ARiZoneSkipArea[FormulaFL] := ARiZoneSkipArea[FormulaFL -1] + ARiZoneAreaInt[FormulaFL -1] + ARiAddArmTime[FormulaFL -1];

END_FOR

IF FormulaFL > iRecipeBlockQty THEN
Step:= 2;
ZoneFL := 1;
GroupFL := 1;
END_IF


2:


FOR ZoneFL:= 1 TO iRecipeBlockQty DO

	FOR GroupFL:= 1 TO 10000 DO

		IF GroupFL > ARiZoneSkipArea[ZoneFL] AND GroupFL <= ARiZoneSkipArea[ZoneFL] + ARiZoneAreaInt[ZoneFL] + ARiAddArmTime[ZoneFL]THEN
		Ar10000_iRecipeTimeBlock [GroupFL] := ARiZoneAddress[ZoneFL];
		END_IF

	END_FOR

END_FOR

IF ZoneFL > iRecipeBlockQty AND GroupFL > 10000 THEN
Step:= 3;
END_IF

3:;


END_CASE
*)
CASE Step2 OF

0:;

1:
iSortMFL:=1;

	IF iSortMFL >0 AND iSortMFL <=iRecipeBlockQty THEN
		FOR iSortMFL := 1 TO iRecipeBlockQty DO

			IF iSortMFL = 1 THEN
			AR2SiRecipeTimeBlock[iSortMFL,1] := 1;
			AR2SiRecipeTimeBlock[iSortMFL,2] := ARiZoneAreaInt[iSortMFL] + ARiAddArmTime[iSortMFL];
			AR2SiRecipeTimeBlock[iSortMFL,3] := ARiZoneAddress[iSortMFL];
			END_IF

			IF iSortMFL > 1 THEN
			AR2SiRecipeTimeBlock[iSortMFL,1] := AR2SiRecipeTimeBlock[iSortMFL-1,2]+1;
			AR2SiRecipeTimeBlock[iSortMFL,2] := ARiZoneAreaInt[iSortMFL] + ARiAddArmTime[iSortMFL] +AR2SiRecipeTimeBlock[iSortMFL-1,2] ;
			AR2SiRecipeTimeBlock[iSortMFL,3] := ARiZoneAddress[iSortMFL];
			END_IF

		END_FOR

	END_IF

IF iSortMFL > iRecipeBlockQty THEN
	Step2:=2;
END_IF


2:
iShiftMFL := 1;
iShiftSFL := 1;

	IF iShiftSFL >0 AND iShiftSFL <=iRecipeBlockQty THEN
		FOR iShiftSFL := 1 TO iRecipeBlockQty DO

			IF AR2SiRecipeTimeBlock[iShiftSFL,2] > AR2SiRecipeTimeBlock[iShiftSFL,1]  THEN
			AR2SiRecipeTimeBlock[iShiftMFL,1] := AR2SiRecipeTimeBlock[iShiftSFL,1];
			AR2SiRecipeTimeBlock[iShiftMFL,2] := AR2SiRecipeTimeBlock[iShiftSFL,2];
			AR2SiRecipeTimeBlock[iShiftMFL,3] := AR2SiRecipeTimeBlock[iShiftSFL,3];

							IF iShiftMFL <> iShiftSFL THEN
							AR2SiRecipeTimeBlock[iShiftSFL,1] := 0;
							AR2SiRecipeTimeBlock[iShiftSFL,2] := 0;
							AR2SiRecipeTimeBlock[iShiftSFL,3] := 0;
							END_IF



			iShiftMFL := iShiftMFL + 1;
			END_IF



		END_FOR

	END_IF


IF iShiftSFL > iRecipeBlockQty THEN
	Step2:=3;
END_IF

3:
iClearRemainFL :=1;

	IF iClearRemainFL >0 AND iClearRemainFL <=iRecipeBlockQty THEN
		FOR iClearRemainFL := 1 TO iRecipeBlockQty DO

			IF AR2SiRecipeTimeBlock[iClearRemainFL,2] <= AR2SiRecipeTimeBlock[iClearRemainFL,1]  THEN
			AR2SiRecipeTimeBlock[iClearRemainFL,1] := 0;
			AR2SiRecipeTimeBlock[iClearRemainFL,2] := 0;
			AR2SiRecipeTimeBlock[iClearRemainFL,3] := 0;
			iShiftMFL := iShiftMFL + 1;
			END_IF

		END_FOR


	END_IF

IF iClearRemainFL > iRecipeBlockQty THEN
Step2:=4;
(*Step2:=5;
bCompleted:=TRUE;
*)
END_IF



4:

iAddMFL:=1;

	IF iAddMFL >0 AND iAddMFL <=iRecipeBlockQty THEN
		FOR iAddMFL := 1 TO iRecipeBlockQty DO
(*
		IF AR2SiRecipeTimeBlock[iAddMFL,3] > iStnQty THEN

			IF iAddMFL = 1 THEN
			AR2SiRecipeTimeBlock[iAddMFL,1] := 1;
			AR2SiRecipeTimeBlock[iAddMFL,2] := ARiZoneAreaInt[iAddMFL] + ARiAddArmTime[iAddMFL];
			AR2SiRecipeTimeBlock[iAddMFL,3] := ARiZoneAddress[iAddMFL];
			END_IF

			IF iAddMFL > 1 THEN
			AR2SiRecipeTimeBlock[iAddMFL,1] := AR2SiRecipeTimeBlock[iAddMFL-1,2]+1;
			AR2SiRecipeTimeBlock[iAddMFL,2] := ARiZoneAreaInt[iAddMFL] + ARiAddArmTime[iAddMFL] +AR2SiRecipeTimeBlock[iAddMFL-1,2] ;
			AR2SiRecipeTimeBlock[iAddMFL,3] := ARiZoneAddress[iAddMFL];
			END_IF

		END_IF
*)
		IF AR2SiRecipeTimeBlock[iAddMFL,3] > 0 AND AR2SiRecipeTimeBlock[iAddMFL,3] <= iStnQty THEN

			IF iAddMFL = 1 THEN
			AR2SiRecipeTimeBlock[iAddMFL,1] := 1;
			AR2SiRecipeTimeBlock[iAddMFL,2] := AR2SiRecipeTimeBlock[iAddMFL+1,2];(*ARiZoneAreaInt[iAddMFL] + ARiAddArmTime[iAddMFL] + ARiZoneAreaInt[iAddMFL+1] ;*)
			AR2SiRecipeTimeBlock[iAddMFL,3] := AR2SiRecipeTimeBlock[iAddMFL,3];
			END_IF

			IF iAddMFL > 1 THEN
			AR2SiRecipeTimeBlock[iAddMFL,1] := AR2SiRecipeTimeBlock[iAddMFL-1,1];
			AR2SiRecipeTimeBlock[iAddMFL,2] := AR2SiRecipeTimeBlock[iAddMFL+1,2];(*ARiZoneAreaInt[iAddMFL] + ARiAddArmTime[iAddMFL] +AR2SiRecipeTimeBlock[iAddMFL-1,2] ;*)
			AR2SiRecipeTimeBlock[iAddMFL,3] := AR2SiRecipeTimeBlock[iAddMFL,3];
			END_IF

		END_IF

		END_FOR

	END_IF

IF iAddMFL > iRecipeBlockQty THEN
	Step2:=5;
bCompleted:=TRUE;
END_IF

5:


;
END_CASE

END_FUNCTION_BLOCK

// ---- FBs/B_JKS_NewFB/FBP-StationRelated/fbMainStationProcess.TcPOU
FUNCTION_BLOCK fbMainStationProcess

VAR_INPUT
	(*fbStnSeqProcess*)
	bSavePB_Uni 									: BOOL; 														(*Universal*) (* Input - HMI - Save Push Button on Touchscreen*)
	bLoadPB_Uni 								: BOOL;														(*Universal*) (* Input - HMI - Load Push Button on Touchscreen*)
	bTrackerEn									: BOOL;														(*During Tracker, it will only call arm when process completed*)
	bTrackerBasedOnPreviousTime			: BOOL;

	(*fbGnrStationMasterController*)
	iCurrentStationAddress_Fix 					: INT;															(*Individual*) (* Input - Define current station no so that this fb know which array number to used*)
	iPreCallArmTime_Uni						: INT;															(*Universal*) (* Input - Pre-Call Arm Time, Program will call arm if the Total process timeEV Equal or Lesser than this value*)
	ARbAlternateStnEn : ARRAY [1..iAlternateSetQty] OF BOOL;
	AR2siAlternateStn : ARRAY [1..iAlternateSetQty, 1..iAlternateStnQty] OF INT;


END_VAR

VAR_IN_OUT PERSISTENT

	(*fbStnSeqProcess*)
(*	DsStnSeqProInput_Ind 						: DS_StnSeqProInput;											(*Individual*) (* Input - PV of Instrument (Temperature, pressure, vacuum and etc), Signal of Sensor to allowed program under the current station status.*)
*)	DSStnSeqProcessCtrl_Ind			 		: DS_fbStnSeqProcessCtrl;									(*Individual*) (* InOut - Link with fbStnSeqProcess, so that this fb know the full status of fbStnSeqProcess and determine which action to take*)

	DsStnSeqRepStore_Ind 						: DS_fbStationSequenceRecipeStore; 						(*Individual*) (* InOut - HMI - The full set of DataStructure-StationSequenceRecipe should selectively display on HMI so that user can customise the recipe by choosing/configure the parameters.*)
	DsStnSubRepStore_Ind 						: DS_fbStationSubRecipeStore; 								(*Individual*) (* InOut - HMI - The full set of DataStructure-StationSubRecipe should selectively display on HMI so that user can customise the recipe by choosing/configure the parameters.*)
	DsStnSeqRepCall_Ind 						: DS_fbStationSequenceRecipeCall;							(*Individual*) (* InOut - Used to call StationSequenceRecipe Detail from fbStationSequenceRecipe*)
	DsStnSubRepCall_Ind 						: DS_fbStationSubRecipeCall;								(*Individual*) (* InOut - Used to call StationSubRecipe Detail from fbStationSubRecipe*)

	(*fbGnrStationMasterController*)
	ARbProductRecipeCallEn_Uni 				: ARRAY [0..iStnQty] OF BOOL;					(*Universal*) (* Output - Link with fbGnrProductRecipeMemory, Array based on Current Station No, the fbGnrProductRecipeMemory will start Read info from Memory when this bool turn on*)
	ARiProductRecipeNoCall_Uni 				: ARRAY [0..iStnQty] OF INT;						(*Universal*) (* Output - Link with fbGnrProductRecipeMemory, Array based on Current Station No, the read out from fbGnrProductRecipeMemory is based on this Product Recipe No*)
	ARiProductRecipeStepCall_Uni 				: ARRAY [0..iStnQty] OF INT;						(*Universal*) (* Output - Link with fbGnrProductRecipeMemory, Array based on Current Station No, the read out from fbGnrProductRecipeMemory is based on this Product Recipe Step No*)

	DSfbGnrProductRecipeMemoryOut_Uni 		: DS_fbGnrProductRecipeMemoryOut;						(*Universal*) (* Input - Link with fbGnrProductRecipeMemory, all the read out info from fbGnrProductRecipeMemory will store in this DataStucture*)

	ARbArmReady_Uni							: ARRAY [1..iArmQty] OF BOOL;								(* Universal*) (* Input  - From ArmPnpFB, This signal is used to confirm if the arm is ready and idling*)

	ARiStnNoToCalledArm_Uni					: ARRAY [0..iArmQty] OF INT; 									(*Universal*) (* Output - Link with fbArmPnP, Array based on Arm No, The Int will store which Station that calling the Arm*)
	ARDSGnrFeedArmPnpParameter_Uni		: ARRAY [0..iArmQty] OF DSGnr_CalledArmPnpParameter; 	(*Universal*) (* Output - Link with fbArmPnP, Array based on Current Station No, Arm should move based on this DataStructure Info*)

	DSLdBasketInfo_Uni		 				: DS_BasketInfo;											(*Input - Loading CONFIRM Basket Info*)
	DSUldBasketInfo_Uni		 				: DS_BasketInfo;											(*Input - Uloading CONFIRM Basket Info*)
	ARDsStnBasketInfo_Uni					: ARRAY [1..iStnQty] OF DS_BasketInfo;						(*Input - Station Basket Info*)



END_VAR

VAR_OUTPUT PERSISTENT
	bSaveInd_Uni 								: BOOL; 														(*Universal*) (* Output - HMI - Save Indicator on Touchscreen*)
	bLoadInd_Uni 								: BOOL; 														(*Universal*) (* Output - HMI - Load Indicator on Touchscreen*)
(*	DSStnSeqProOutput_Ind 						:DS_StnSeqProOutput;										(*Individual*) (* Output - To Control Output - When process running, instrument should control by the output in this Data structure*)
*)
END_VAR



VAR PERSISTENT
	(*fbStnSeqProcess*)
	StnSeqProcessfb: fbStnSeqProcess;
	bStnSeqProcessStartInterlock			: BOOL;															(*Individual*) (* Input - Interlocking to Enable the StnSeqProcess Start Signal, It might used on those station with Sliding door for close confirmation before process start*)

	(*fbGnrStationMasterController*)
	GnrStationMasterControllerfb				: fbGnrStationMasterController;
	bStnSeqProcessSt						: BOOL;															(* Output - Link with fbStnSeqProcess, After Read out from fbGnrProductRecipeMemory, this fb will trigger this Bool to start the StnSeqProcess*)
	DSGnrBufferCalledArmPnpParameter 	: DSGnr_CalledArmPnpParameter;								(* Internal used, Buffer Data Structure read out from fbGnrProductRecipeMemory*)
	DSGnrBuffersPnpSequenceDescription	: STRING (99);														(* Internal used, Buffer Description read out from fbGnrProductRecipeMemory*)
	ARiPreviousStnSeqTotalProcessTime 	: ARRAY [0..iProductRecipeArrayQty] OF INT;					(* Internal used, Previous Total Process Time will save into this Array, Array based on StationSequenceNo*)
	iCallStep									: INT;																(* Internal used, to monitor the current Step so that you can indentify the error of this function block if stucked*)
	DSBasketInfo_Ind 							: DS_BasketInfo;												(*Individual*) (* InOut - Basket Information that comes into current station*)

END_VAR
VAR
	bLdStnConfirm: BOOL;
	bUldStnConfirm: BOOL;
	bStn1Confirm: BOOL;
	bGreaterStn1Confirm: BOOL;
	bLesserStnQtyConfirm: BOOL;
	bEqualStnQtyConfirm: BOOL;
	iTotalProcessTimeSV: INT;
END_VAR
VAR // added by the converter: edge detectors and wires of the graphical bodies
    _w1, _w2, _w3 : DS_BasketInfo;
END_VAR

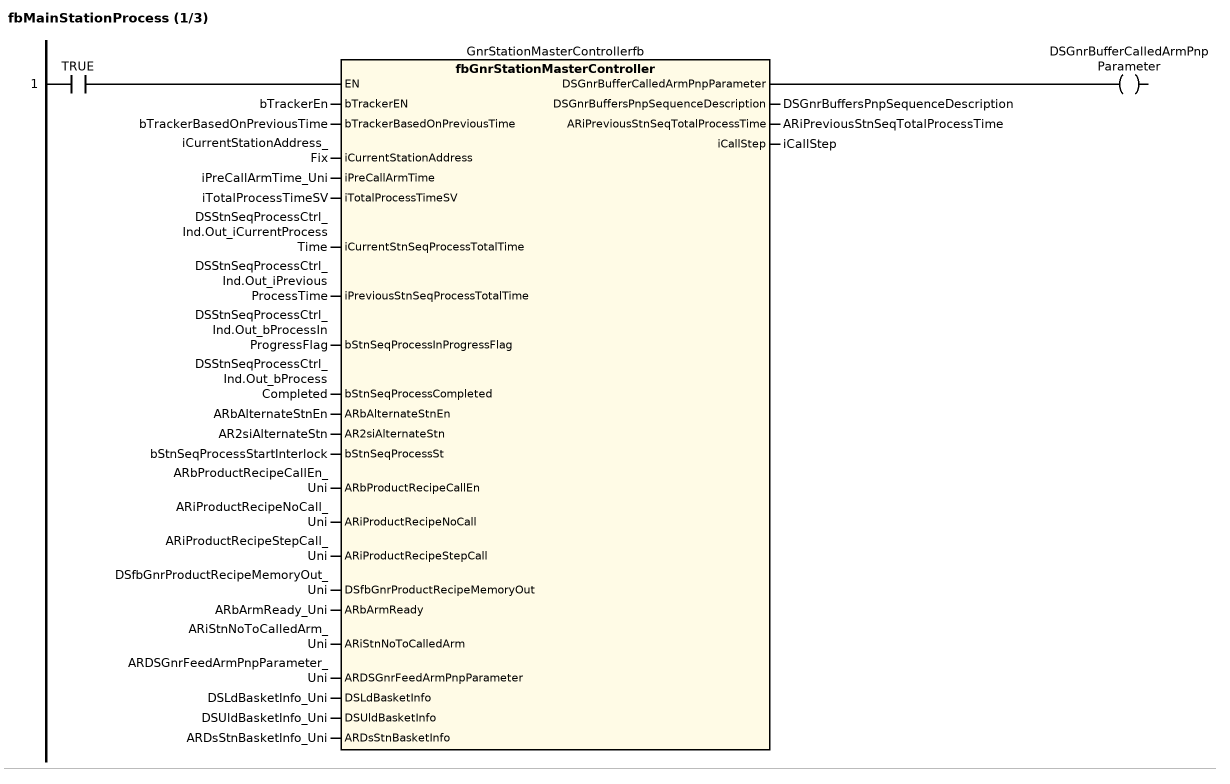
// NETWORK 1
GnrStationMasterControllerfb(
    bTrackerEN := bTrackerEn,
    bTrackerBasedOnPreviousTime := bTrackerBasedOnPreviousTime,
    iCurrentStationAddress := iCurrentStationAddress_Fix,
    iPreCallArmTime := iPreCallArmTime_Uni,
    iTotalProcessTimeSV := iTotalProcessTimeSV,
    iCurrentStnSeqProcessTotalTime := DSStnSeqProcessCtrl_Ind.Out_iCurrentProcessTime,
    iPreviousStnSeqProcessTotalTime := DSStnSeqProcessCtrl_Ind.Out_iPreviousProcessTime,
    bStnSeqProcessInProgressFlag := DSStnSeqProcessCtrl_Ind.Out_bProcessInProgressFlag,
    bStnSeqProcessCompleted := DSStnSeqProcessCtrl_Ind.Out_bProcessCompleted,
    ARbAlternateStnEn := ARbAlternateStnEn,
    AR2siAlternateStn := AR2siAlternateStn,
    bStnSeqProcessSt := bStnSeqProcessStartInterlock,
    ARbProductRecipeCallEn := ARbProductRecipeCallEn_Uni,
    ARiProductRecipeNoCall := ARiProductRecipeNoCall_Uni,
    ARiProductRecipeStepCall := ARiProductRecipeStepCall_Uni,
    DSfbGnrProductRecipeMemoryOut := DSfbGnrProductRecipeMemoryOut_Uni,
    ARbArmReady := ARbArmReady_Uni,
    ARiStnNoToCalledArm := ARiStnNoToCalledArm_Uni,
    ARDSGnrFeedArmPnpParameter := ARDSGnrFeedArmPnpParameter_Uni,
    DSLdBasketInfo := DSLdBasketInfo_Uni,
    DSUldBasketInfo := DSUldBasketInfo_Uni,
    ARDsStnBasketInfo := ARDsStnBasketInfo_Uni,
    DSGnrBuffersPnpSequenceDescription => DSGnrBuffersPnpSequenceDescription,
    ARiPreviousStnSeqTotalProcessTime => ARiPreviousStnSeqTotalProcessTime,
    iCallStep => iCallStep); // fbGnrStationMasterController
DSGnrBufferCalledArmPnpParameter := GnrStationMasterControllerfb.DSGnrBufferCalledArmPnpParameter;

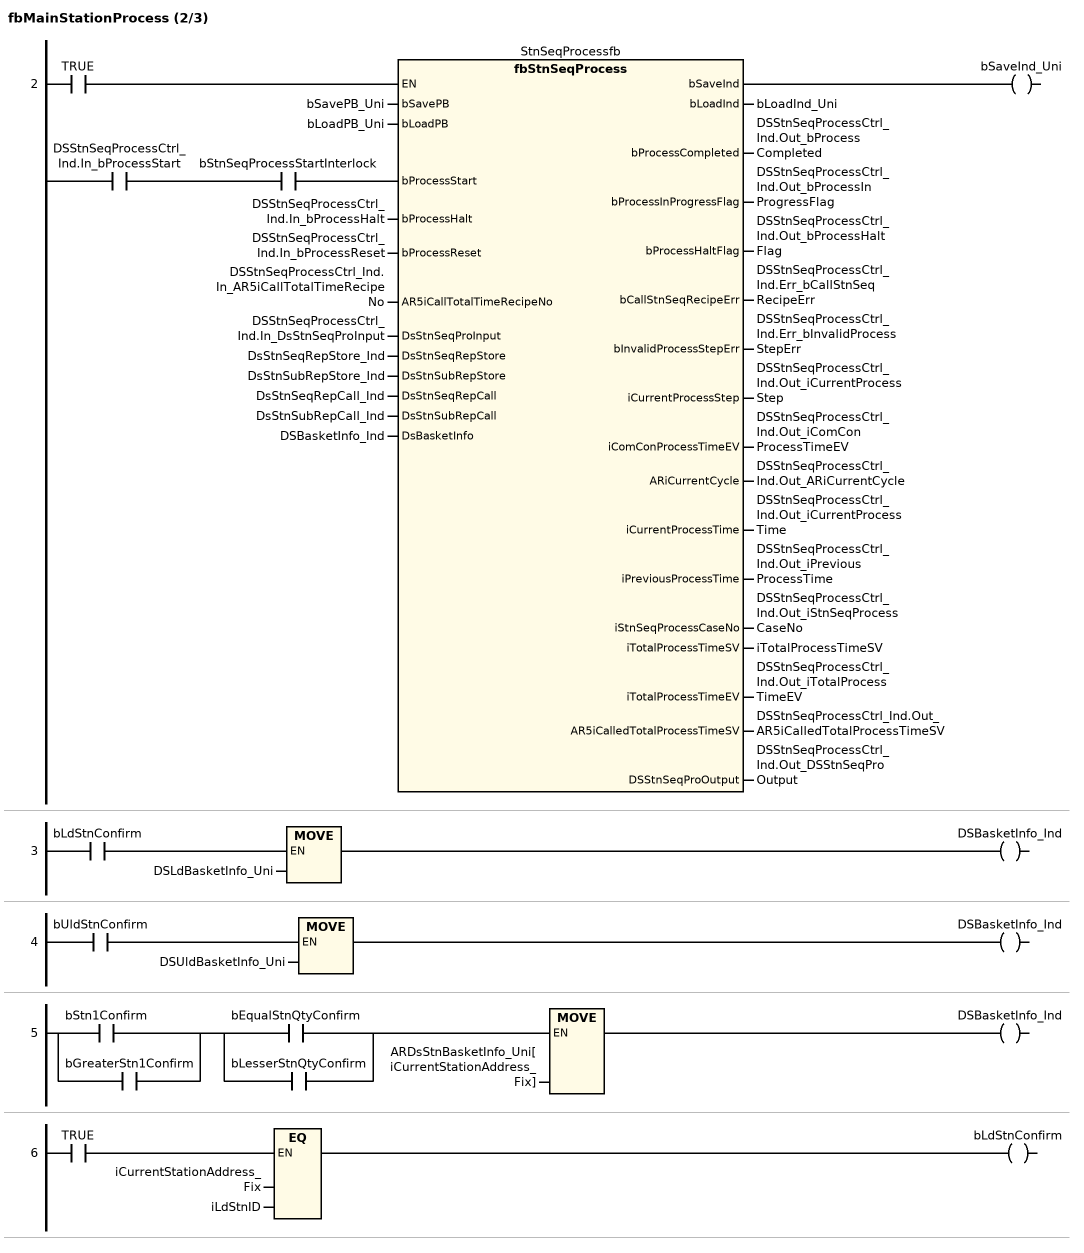
// NETWORK 2
StnSeqProcessfb(
    bSavePB := bSavePB_Uni,
    bLoadPB := bLoadPB_Uni,
    bProcessStart := DSStnSeqProcessCtrl_Ind.In_bProcessStart AND bStnSeqProcessStartInterlock,
    bProcessHalt := DSStnSeqProcessCtrl_Ind.In_bProcessHalt,
    bProcessReset := DSStnSeqProcessCtrl_Ind.In_bProcessReset,
    AR5iCallTotalTimeRecipeNo := DSStnSeqProcessCtrl_Ind.In_AR5iCallTotalTimeRecipeNo,
    DsStnSeqProInput := DSStnSeqProcessCtrl_Ind.In_DsStnSeqProInput,
    DsStnSeqRepStore := DsStnSeqRepStore_Ind,
    DsStnSubRepStore := DsStnSubRepStore_Ind,
    DsStnSeqRepCall := DsStnSeqRepCall_Ind,
    DsStnSubRepCall := DsStnSubRepCall_Ind,
    DsBasketInfo := DSBasketInfo_Ind,
    bLoadInd => bLoadInd_Uni,
    bProcessCompleted => DSStnSeqProcessCtrl_Ind.Out_bProcessCompleted,
    bProcessInProgressFlag => DSStnSeqProcessCtrl_Ind.Out_bProcessInProgressFlag,
    bProcessHaltFlag => DSStnSeqProcessCtrl_Ind.Out_bProcessHaltFlag,
    bCallStnSeqRecipeErr => DSStnSeqProcessCtrl_Ind.Err_bCallStnSeqRecipeErr,
    bInvalidProcessStepErr => DSStnSeqProcessCtrl_Ind.Err_bInvalidProcessStepErr,
    iCurrentProcessStep => DSStnSeqProcessCtrl_Ind.Out_iCurrentProcessStep,
    iComConProcessTimeEV => DSStnSeqProcessCtrl_Ind.Out_iComConProcessTimeEV,
    ARiCurrentCycle => DSStnSeqProcessCtrl_Ind.Out_ARiCurrentCycle,
    iCurrentProcessTime => DSStnSeqProcessCtrl_Ind.Out_iCurrentProcessTime,
    iPreviousProcessTime => DSStnSeqProcessCtrl_Ind.Out_iPreviousProcessTime,
    iStnSeqProcessCaseNo => DSStnSeqProcessCtrl_Ind.Out_iStnSeqProcessCaseNo,
    iTotalProcessTimeSV => iTotalProcessTimeSV,
    iTotalProcessTimeEV => DSStnSeqProcessCtrl_Ind.Out_iTotalProcessTimeEV,
    AR5iCalledTotalProcessTimeSV => DSStnSeqProcessCtrl_Ind.Out_AR5iCalledTotalProcessTimeSV,
    DSStnSeqProOutput => DSStnSeqProcessCtrl_Ind.Out_DSStnSeqProOutput); // fbStnSeqProcess
bSaveInd_Uni := StnSeqProcessfb.bSaveInd;

// NETWORK 3
IF bLdStnConfirm THEN _w1 := DSLdBasketInfo_Uni; END_IF
DSBasketInfo_Ind := _w1;

// NETWORK 4
IF bUldStnConfirm THEN _w2 := DSUldBasketInfo_Uni; END_IF
DSBasketInfo_Ind := _w2;

// NETWORK 5
IF (bStn1Confirm OR bGreaterStn1Confirm) AND (bEqualStnQtyConfirm OR bLesserStnQtyConfirm) THEN
    _w3 := ARDsStnBasketInfo_Uni[iCurrentStationAddress_Fix];
END_IF
DSBasketInfo_Ind := _w3;

// NETWORK 6
bLdStnConfirm := iCurrentStationAddress_Fix = iLdStnID;

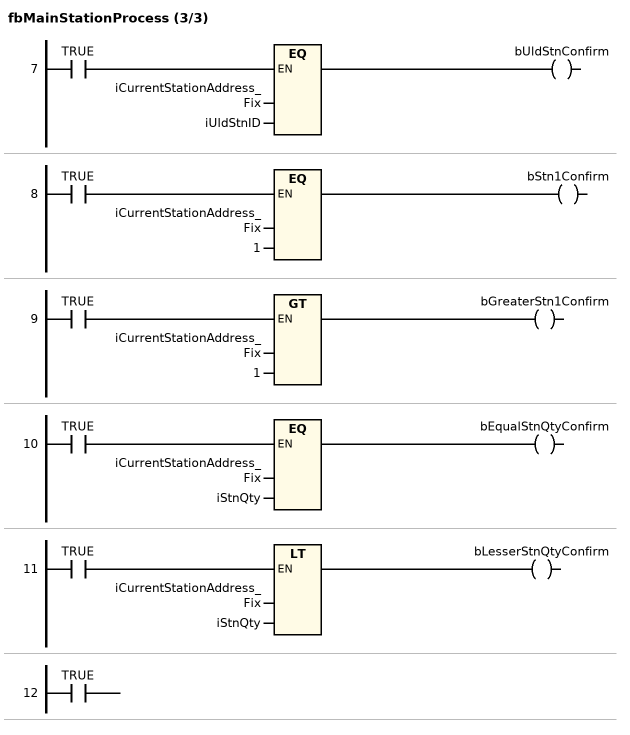
// NETWORK 7
bUldStnConfirm := iCurrentStationAddress_Fix = iUldStnID;

// NETWORK 8
bStn1Confirm := iCurrentStationAddress_Fix = 1;

// NETWORK 9
bGreaterStn1Confirm := iCurrentStationAddress_Fix > 1;

// NETWORK 10
bEqualStnQtyConfirm := iCurrentStationAddress_Fix = iStnQty;

// NETWORK 11
bLesserStnQtyConfirm := iCurrentStationAddress_Fix < iStnQty;

// NETWORK 12

END_FUNCTION_BLOCK

// ---- FBs/B_JKS_NewFB/FBP-TempController/fbTempControl.TcPOU
FUNCTION_BLOCK fbTempControl
VAR_INPUT
	iRawAnalogInput					: INT;
	rRawToPVRatio					: REAL;
	rTargetTempHysteresis			: REAL;
	rBasedHighTempSV				: REAL;
	rBasedTargetTempSV				: REAL;
	rBasedTempReadySV				: REAL;
	rBased1stLimitSV					: REAL;
(*	rBased2ndLimitSV					: REAL;*)
	rOverrideTargetTempSV			: REAL;
	rOverrideTempReadySV			: REAL;
	rOverride1stLimitSV				: REAL;
(*	rOverride2ndLimitSV				: REAL;*)

	bTemperatureOverrideEn			: BOOL;
	bManualHeaterOnPB				: BOOL;
	bPreparation						: BOOL;
	bAutoStart						: BOOL;
	bDeactivatedMode				: BOOL;
	iNotReadyAlarmDelayTime					: INT;

END_VAR
VAR_OUTPUT
	rTemperaturePV				: REAL;
	bOutputHeater				: BOOL;
	bStatusTempReadyNO					: BOOL;
	bAlarmHighTempNC					: BOOL;
	bAlarm1stLimitNO					: BOOL;
	bAlarmTemperatureNotReady 		: BOOL;
(*	bAlarm2ndLimit					: BOOL;
	b_ConditionNotFullfill	: BOOL;
	b_TempNotRdyAlarm	: BOOL;*)

END_VAR
VAR
	rInternalTempRdyPlus: REAL;
	rInternalTempRdyMinus: REAL;
	rInternalTempHysPlus: REAL;
	rInternalTempHysMinus: REAL;
	rInternal1stLimitPlus: REAL;
	rInternal1stLimitMinus: REAL;
	rInternalTargetTempSV : REAL;
(*	rInternal2ndLimitPlus: REAL;
	rInternal2ndLimitMinus: REAL;*)
(*	tPowerOnDelayTimer: TON;
	tPowerOnDelayTimer_RE: R_TRIG;
*)	tNotReadyAlarmDelayTimer: TON;
	bManualHeaterOnPB_RE: R_TRIG;
	bPreparation_RE: R_TRIG;
	bAutoStart_RE: R_TRIG;
END_VAR

(*tPowerOnDelayTimer(IN:=TRUE, PT:=t#1s , Q=> , ET=> );
tPowerOnDelayTimer_RE(CLK:=tPowerOnDelayTimer.Q , Q=> );
*)

IF rRawToPVRatio <> 0 AND iRawAnalogInput > 0 THEN
rTemperaturePV := INT_TO_REAL(iRawAnalogInput)/rRawToPVRatio ;
ELSE
rTemperaturePV := 0 ;
END_IF

IF bTemperatureOverrideEn THEN

	rInternalTargetTempSV := rOverrideTargetTempSV;
	rInternalTempRdyPlus := rOverrideTargetTempSV+rOverrideTempReadySV;
	rInternalTempRdyMinus := rOverrideTargetTempSV-rOverrideTempReadySV;

	rInternalTempHysPlus :=rOverrideTargetTempSV+ rTargetTempHysteresis;
	rInternalTempHysMinus := rOverrideTargetTempSV-rTargetTempHysteresis;

	rInternal1stLimitPlus := rOverrideTargetTempSV+rOverride1stLimitSV;
	rInternal1stLimitMinus := rOverrideTargetTempSV-rOverride1stLimitSV;
(*
	rInternal2ndLimitPlus := rOverrideTargetTempSV+rOverride2ndLimitSV;
	rInternal2ndLimitMinus := rOverrideTargetTempSV-rOverride2ndLimitSV;
*)
ELSE

	rInternalTargetTempSV := rBasedTargetTempSV;
	rInternalTempRdyPlus := rBasedTargetTempSV+rBasedTempReadySV;
	rInternalTempRdyMinus := rBasedTargetTempSV-rBasedTempReadySV;

	rInternalTempHysPlus := rBasedTargetTempSV+ rTargetTempHysteresis;
	rInternalTempHysMinus := rBasedTargetTempSV-rTargetTempHysteresis;

	rInternal1stLimitPlus := rBasedTargetTempSV+rBased1stLimitSV;
	rInternal1stLimitMinus := rBasedTargetTempSV-rBased1stLimitSV;
(*
	rInternal2ndLimitPlus := rBasedTargetTempSV+rBased2ndLimitSV;
	rInternal2ndLimitMinus := rBasedTargetTempSV-rBased2ndLimitSV;
*)
END_IF
(*
IF  bAutoStart AND (rTemperaturePV >= rInternal2ndLimitPlus OR rTemperaturePV <= rInternal2ndLimitMinus) THEN
	bAlarm2ndLimit := TRUE;
ELSE
	bAlarm2ndLimit := FALSE;
END_IF
*)
IF bAutoStart AND (rTemperaturePV >= rInternal1stLimitPlus OR rTemperaturePV <= rInternal1stLimitMinus) AND NOT bDeactivatedMode THEN
	bAlarm1stLimitNO := TRUE;
ELSE
	bAlarm1stLimitNO := FALSE;
END_IF

IF rTemperaturePV >= rInternalTempRdyMinus AND rTemperaturePV <= rInternalTempRdyPlus THEN
	bStatusTempReadyNO	:= TRUE;
ELSE
	bStatusTempReadyNO	:= FALSE;
END_IF



(*Heater Output Control*)
bManualHeaterOnPB_RE(CLK:=bManualHeaterOnPB , Q=> );
bPreparation_RE(CLK:=bPreparation , Q=> );
bAutoStart_RE(CLK:=bAutoStart , Q=> );



IF rTemperaturePV >= rInternalTargetTempSV OR bDeactivatedMode THEN
	bOutputHeater := FALSE;
ELSIF  rTemperaturePV <= rInternalTempHysMinus AND bAlarmHighTempNC  THEN
	bOutputHeater := TRUE;
ELSIF rTemperaturePV < rInternalTargetTempSV AND (bManualHeaterOnPB_RE.Q OR bPreparation_RE.Q AND bAutoStart_RE.Q)   AND bAlarmHighTempNC THEN
	bOutputHeater := TRUE;
END_IF

tNotReadyAlarmDelayTimer(IN:=NOT bStatusTempReadyNO AND bPreparation AND NOT bAutoStart , PT:= INT_TO_TIME(iNotReadyAlarmDelayTime*1000) , Q=> , ET=> );
IF  tNotReadyAlarmDelayTimer.Q THEN
bAlarmTemperatureNotReady := TRUE;
ELSE
bAlarmTemperatureNotReady := FALSE;
END_IF


IF rTemperaturePV >= rBasedHighTempSV AND NOT bDeactivatedMode THEN
	bAlarmHighTempNC := FALSE;
ELSE
	bAlarmHighTempNC := TRUE;
END_IF

END_FUNCTION_BLOCK

// ---- FBs/B_JKS_NewFB_V2/FBP-ArmRelated/fbV2_ArmPosSignalCtrl.TcPOU
FUNCTION_BLOCK fbV2_ArmPosSignalCtrl

VAR_INPUT
	bHomeDone 								: BOOL;
	bVertMovementEn							: BOOL;
	bHorzMovementEn						: BOOL;
	bDisableHorzCheckForVerticalPos			: BOOL;
	lrCurrentPos								: LREAL;
	lrTargetPos								: LREAL;
	lrPosCfmTolerance						: LREAL;
	lr2ndSpdRange							: LREAL;
	tPositionCfmDelayOnTime					: TIME;

	ARbLdHorzZoneConfirm 		: ARRAY [0..iLdStnQty] OF BOOL; (*From fbV2_FBPArmHorzZoneConfirm*)
	ARbHorzStnZoneConfirm 		: ARRAY [1..iStnQty] OF BOOL; (*From fbV2_FBPArmHorzZoneConfirm*)
	ARbUldHorzZoneConfirm 		: ARRAY [0..iUldStnQty] OF BOOL; (*From fbV2_FBPArmHorzZoneConfirm*)

(*
	lrHorz_CurrentPos								: LREAL;
	lrHorz_TargetPos								: LREAL;
	lrHorz_PosCfmTolerance						: LREAL;
	lrHorz_2ndSpdRange							: LREAL;
*)
END_VAR

VAR_OUTPUT
	lrPosToleranceP : ARRAY [0..3, 0..iStnQty, 0..12] OF LREAL;
	lrPosToleranceN : ARRAY [0..3, 0..iStnQty, 0..12] OF LREAL;

END_VAR

VAR_IN_OUT PERSISTENT

	DSArmPosition 					: DSV2_ArmPosition;
END_VAR



VAR PERSISTENT



	lrPos2ndSpdP : ARRAY [0..3, 0..iStnQty, 0..12] OF LREAL;
	lrPos2ndSpdN : ARRAY [0..3, 0..iStnQty, 0..12] OF LREAL;

	ARtDelayTimer : ARRAY [0..3, 0..iStnQty, 0..12] OF TON;

(*
	ARlrBufferLdHookPosToleranceP			: ARRAY [0..iLdStnQty] OF LREAL;
	ARlrBufferLdUnhookPosToleranceP			: ARRAY [0..iLdStnQty] OF LREAL;
	ARlrBufferUldHookPosToleranceP			: ARRAY [0..iUldStnQty] OF LREAL;
	ARlrBufferUldUnhookPosToleranceP			: ARRAY [0..iUldStnQty] OF LREAL;

	ARlrBufferStnHookPosToleranceP			: ARRAY [0..iStnQty] OF LREAL;
	ARlrBufferStnUnhookPosToleranceP			: ARRAY [0..iStnQty] OF LREAL;

	iToleranceN: INT;

	ARlrBufferLdHookPosToleranceN			: ARRAY [0..iLdStnQty] OF LREAL;
	ARlrBufferLdUnhookPosToleranceN			: ARRAY [0..iLdStnQty] OF LREAL;
	ARlrBufferUldHookPosToleranceN			: ARRAY [0..iUldStnQty] OF LREAL;
	ARlrBufferUldUnhookPosToleranceN		: ARRAY [0..iUldStnQty] OF LREAL;

	ARlrBufferStnHookPosToleranceN			: ARRAY [0..iStnQty] OF LREAL;
	ARlrBufferStnUnhookPosToleranceN			: ARRAY [0..iStnQty] OF LREAL;

	i2ndSpdP: INT;

	ARlrBufferLdHookPos2ndSpdP				: ARRAY [0..iLdStnQty] OF LREAL;
	ARlrBufferLdUnhookPos2ndSpdP			: ARRAY [0..iLdStnQty] OF LREAL;
	ARlrBufferUldHookPos2ndSpdP				: ARRAY [0..iUldStnQty] OF LREAL;
	ARlrBufferUldUnhookPos2ndSpdP			: ARRAY [0..iUldStnQty] OF LREAL;

	ARlrBufferStnHookPos2ndSpdP				: ARRAY [0..iStnQty] OF LREAL;
	ARlrBufferStnUnhookPos2ndSpdP			: ARRAY [0..iStnQty] OF LREAL;

	i2ndSpdN: INT;

	ARlrBufferLdHookPos2ndSpdN				: ARRAY [0..iLdStnQty] OF LREAL;
	ARlrBufferLdUnhookPos2ndSpdN			: ARRAY [0..iLdStnQty] OF LREAL;
	ARlrBufferUldHookPos2ndSpdN				: ARRAY [0..iUldStnQty] OF LREAL;
	ARlrBufferUldUnhookPos2ndSpdN			: ARRAY [0..iUldStnQty] OF LREAL;

	ARlrBufferStnHookPos2ndSpdN				: ARRAY [0..iStnQty] OF LREAL;
	ARlrBufferStnUnhookPos2ndSpdN			: ARRAY [0..iStnQty] OF LREAL;
*)
END_VAR

VAR

	iSFLQty: INT;

	iGenFL1: INT;
	iGenFL2: INT;
	iGenFL3: INT;

	iSignalFL1: INT;
	iSignalFL2: INT;
	iSignalFL3: INT;
END_VAR

(*
Stage 1 --> (0..3) 
------------------------
1=Stn
2=Loading
3=Unloading


Stage 2 --> (0..iStnQty) 
------------------------
No = Station No (Example: 8 = Station 8)



Stage 3 --> (0..12) 
------------------------
1=Vert - Up
2=Vert - SlowPull / Slanted
3=Vert - Regular / Mid Top
4=Vert - AgiUp
5=Vert - AgiDown
6=Vert - Down
7=Horz - Unhook 
8=Horz -  Hook
9=Horz -  Slanted Left
10=Horz - Slanted Right
11=Reserved
12=Reserved
*)

(* Generate Positive/Negative Tolerance and Positive/Negative 2nd Speed  *)
(*[][][][][][][][][][][][][][][][][][][][][][][][][][][][][][][][][][][][][][][][][][][][][][][][][][][][][][][][][][][][][][][][][][][][][][][][][][][][][][][][][][][][][][][][][][][][][][][][][][][]*)

iGenFL1 := 1;

FOR iGenFL1 := 1 TO 3 DO
	IF iGenFL1 >= 1 AND iGenFL1 <= 3 THEN

		IF iGenFL1 = 1 THEN
		iSFLQty := iStnQty;
		ELSIF iGenFL1 = 2 THEN
		iSFLQty := iLdStnQty;
		ELSIF iGenFL1 = 3 THEN
		iSFLQty := iUldStnQty;
		END_IF

		iGenFL2 := 1;

		FOR iGenFL2 := 1 TO iSFLQty DO
			IF iGenFL2 >= 1 AND iGenFL2 <= iSFLQty THEN

				iGenFL3 := 1;

				FOR iGenFL3 := 1 TO 12 DO
					IF iGenFL3 >= 1 AND iGenFL3 <= 12 THEN


						IF iGenFL3 >= 1 AND iGenFL3 <= 6 AND bVertMovementEn AND NOT bHorzMovementEn THEN
						lrPosToleranceP[iGenFL1, iGenFL2, iGenFL3] := DSArmPosition.AR3slrPosition[iGenFL1, iGenFL2, iGenFL3]+lrPosCfmTolerance;
						lrPosToleranceN[iGenFL1, iGenFL2, iGenFL3] := DSArmPosition.AR3slrPosition[iGenFL1, iGenFL2, iGenFL3]-lrPosCfmTolerance;

						lrPos2ndSpdP[iGenFL1, iGenFL2, iGenFL3] := DSArmPosition.AR3slrPosition[iGenFL1, iGenFL2, iGenFL3]+lr2ndSpdRange;
						lrPos2ndSpdN[iGenFL1, iGenFL2, iGenFL3] := DSArmPosition.AR3slrPosition[iGenFL1, iGenFL2, iGenFL3]-lr2ndSpdRange;
						END_IF

						IF iGenFL3 >= 7 AND iGenFL3 <= 10 AND bHorzMovementEn AND NOT bVertMovementEn THEN
						lrPosToleranceP[iGenFL1, iGenFL2, iGenFL3] := DSArmPosition.AR3slrPosition[iGenFL1, iGenFL2, iGenFL3]+lrPosCfmTolerance;
						lrPosToleranceN[iGenFL1, iGenFL2, iGenFL3] := DSArmPosition.AR3slrPosition[iGenFL1, iGenFL2, iGenFL3]-lrPosCfmTolerance;

						lrPos2ndSpdP[iGenFL1, iGenFL2, iGenFL3] := DSArmPosition.AR3slrPosition[iGenFL1, iGenFL2, iGenFL3]+lr2ndSpdRange;
						lrPos2ndSpdN[iGenFL1, iGenFL2, iGenFL3] := DSArmPosition.AR3slrPosition[iGenFL1, iGenFL2, iGenFL3]-lr2ndSpdRange;
						END_IF

					END_IF
				END_FOR
			END_IF
		END_FOR
	END_IF
END_FOR



(*
(*Generate Pos Confirm Bit and  2nd Speed Bit*)
(*[][][][][][][][][][][][][][][][][][][][][][][][][][][][][][][][][][][][][][][][][][][][][][][][][][][][][][][][][][][][][][][][][][][][][][][][][][][][][][][][][][][][][][][][][][][][][][][][][][][]*)

iSignalFL1 := 1;

FOR iSignalFL1 := 1 TO 3 DO
	IF iSignalFL1 >= 1 AND iSignalFL1 <= 3 THEN

		IF iSignalFL1 = 1 THEN
		iSFLQty := iStnQty;
		ELSIF iSignalFL1 = 2 THEN
		iSFLQty := iLdStnQty;
		ELSIF iSignalFL1 = 3 THEN
		iSFLQty := iUldStnQty;
		END_IF

		iSignalFL2 := 1;

		FOR iSignalFL2 := 1 TO iSFLQty DO
			IF iSignalFL2 >= 1 AND iSignalFL2 <= iSFLQty THEN

				iSignalFL3 := 1;

				FOR iSignalFL3 := 1 TO 12 DO
					IF iSignalFL3 >= 1 AND iSignalFL3 <= 12 THEN

						IF DSArmPosition.AR3slrPosition[iSignalFL1, iSignalFL2, iSignalFL3] <> 0 THEN

							IF (iSignalFL3 >= 1 AND iSignalFL3 <= 6 AND bVertMovementEn AND NOT bHorzMovementEn)
							OR (iSignalFL3 >= 7 AND iSignalFL3 <= 10 AND bHorzMovementEn AND NOT bVertMovementEn) THEN

								IF lrCurrentPos >= lrPos2ndSpdN[iSignalFL1, iSignalFL2, iSignalFL3]  AND lrCurrentPos <= lrPos2ndSpdP[iSignalFL1, iSignalFL2, iSignalFL3] AND lrTargetPos = DSArmPosition.AR3slrPosition[iSignalFL1,iSignalFL2,iSignalFL3] AND bHomeDone THEN
								DSArmPosition.AR3sb2ndSpdEn[iSignalFL1,iSignalFL2,iSignalFL3] := TRUE;
								ELSE
								DSArmPosition.AR3sb2ndSpdEn[iSignalFL1,iSignalFL2,iSignalFL3] := FALSE;
								END_IF

							END_IF

							IF (iSignalFL3 >= 7 AND iSignalFL3 <= 10 AND bHorzMovementEn AND NOT bVertMovementEn)
							OR (iSignalFL3 = 1 AND bVertMovementEn AND NOT bHorzMovementEn) THEN

									IF lrCurrentPos >= lrPosToleranceN[iSignalFL1, iSignalFL2, iSignalFL3]  AND lrCurrentPos <= lrPosToleranceP[iSignalFL1, iSignalFL2, iSignalFL3] AND bHomeDone THEN
									DSArmPosition.AR3sbPositionCfm[iSignalFL1,iSignalFL2,iSignalFL3] := TRUE;
									ELSE
									DSArmPosition.AR3sbPositionCfm[iSignalFL1,iSignalFL2,iSignalFL3] := FALSE;
									END_IF

							ELSIF (iSignalFL3 >= 2 AND iSignalFL3 <= 6 AND bVertMovementEn AND NOT bHorzMovementEn) THEN

								IF ((iSignalFL1 = 1 AND ARbHorzStnZoneConfirm[iSignalFL2])
								OR (iSignalFL1 = 2 AND ARbLdHorzZoneConfirm[iSignalFL2])
								OR (iSignalFL1 = 3 AND ARbUldHorzZoneConfirm[iSignalFL2])) OR bDisableHorzCheckForVerticalPos  THEN
									IF lrCurrentPos >= lrPosToleranceN[iSignalFL1, iSignalFL2, iSignalFL3]  AND lrCurrentPos <= lrPosToleranceP[iSignalFL1, iSignalFL2, iSignalFL3] AND bHomeDone THEN
									DSArmPosition.AR3sbPositionCfm[iSignalFL1,iSignalFL2,iSignalFL3] := TRUE;
									ELSE
									DSArmPosition.AR3sbPositionCfm[iSignalFL1,iSignalFL2,iSignalFL3] := FALSE;
									END_IF
								ELSE
								DSArmPosition.AR3sbPositionCfm[iSignalFL1,iSignalFL2,iSignalFL3] := FALSE;
								END_IF
							END_IF




						ELSE
							DSArmPosition.AR3sbPositionCfm[iSignalFL1,iSignalFL2,iSignalFL3] := FALSE;
							DSArmPosition.AR3sb2ndSpdEn[iSignalFL1,iSignalFL2,iSignalFL3] := FALSE;
						END_IF

					END_IF
				END_FOR
			END_IF
		END_FOR
	END_IF
END_FOR
*)


(*Generate Pos Confirm Bit and  2nd Speed Bit*)
(*[][][][][][][][][][][][][][][][][][][][][][][][][][][][][][][][][][][][][][][][][][][][][][][][][][][][][][][][][][][][][][][][][][][][][][][][][][][][][][][][][][][][][][][][][][][][][][][][][][][]*)

iSignalFL1 := 1;

FOR iSignalFL1 := 1 TO 3 DO
	IF iSignalFL1 >= 1 AND iSignalFL1 <= 3 THEN

		IF iSignalFL1 = 1 THEN
		iSFLQty := iStnQty;
		ELSIF iSignalFL1 = 2 THEN
		iSFLQty := iLdStnQty;
		ELSIF iSignalFL1 = 3 THEN
		iSFLQty := iUldStnQty;
		END_IF

		iSignalFL2 := 1;

		FOR iSignalFL2 := 1 TO iSFLQty DO
			IF iSignalFL2 >= 1 AND iSignalFL2 <= iSFLQty THEN

				iSignalFL3 := 1;

				FOR iSignalFL3 := 1 TO 12 DO
					IF iSignalFL3 >= 1 AND iSignalFL3 <= 12 THEN

						IF DSArmPosition.AR3slrPosition[iSignalFL1, iSignalFL2, iSignalFL3] <> 0 THEN

							IF (iSignalFL3 >= 1 AND iSignalFL3 <= 6 AND bVertMovementEn AND NOT bHorzMovementEn)
							OR (iSignalFL3 >= 7 AND iSignalFL3 <= 10 AND bHorzMovementEn AND NOT bVertMovementEn) THEN
								IF lrCurrentPos >= lrPos2ndSpdN[iSignalFL1, iSignalFL2, iSignalFL3]  AND lrCurrentPos <= lrPos2ndSpdP[iSignalFL1, iSignalFL2, iSignalFL3] AND lrTargetPos = DSArmPosition.AR3slrPosition[iSignalFL1,iSignalFL2,iSignalFL3] AND bHomeDone THEN
								DSArmPosition.AR3sb2ndSpdEn[iSignalFL1,iSignalFL2,iSignalFL3] := TRUE;
								ELSE
								DSArmPosition.AR3sb2ndSpdEn[iSignalFL1,iSignalFL2,iSignalFL3] := FALSE;
								END_IF

							END_IF

							IF (iSignalFL3 >= 7 AND iSignalFL3 <= 10 AND bHorzMovementEn AND NOT bVertMovementEn)
							OR (iSignalFL3 = 1 AND bVertMovementEn AND NOT bHorzMovementEn) THEN

									ARtDelayTimer[iSignalFL1,iSignalFL2,iSignalFL3](IN:=
									lrCurrentPos >= lrPosToleranceN[iSignalFL1, iSignalFL2, iSignalFL3]  AND lrCurrentPos <= lrPosToleranceP[iSignalFL1, iSignalFL2, iSignalFL3] AND bHomeDone ,
									PT:=tPositionCfmDelayOnTime , Q=> , ET=> );

									IF ARtDelayTimer[iSignalFL1,iSignalFL2,iSignalFL3].Q THEN
									DSArmPosition.AR3sbPositionCfm[iSignalFL1,iSignalFL2,iSignalFL3] := TRUE;
									ELSE
									DSArmPosition.AR3sbPositionCfm[iSignalFL1,iSignalFL2,iSignalFL3] := FALSE;
									END_IF

							ELSIF (iSignalFL3 >= 2 AND iSignalFL3 <= 6 AND bVertMovementEn AND NOT bHorzMovementEn) THEN

								IF ((iSignalFL1 = 1 AND ARbHorzStnZoneConfirm[iSignalFL2])
								OR (iSignalFL1 = 2 AND ARbLdHorzZoneConfirm[iSignalFL2])
								OR (iSignalFL1 = 3 AND ARbUldHorzZoneConfirm[iSignalFL2])) OR bDisableHorzCheckForVerticalPos  THEN

									ARtDelayTimer[iSignalFL1,iSignalFL2,iSignalFL3](IN:=
									lrCurrentPos >= lrPosToleranceN[iSignalFL1, iSignalFL2, iSignalFL3]  AND lrCurrentPos <= lrPosToleranceP[iSignalFL1, iSignalFL2, iSignalFL3] AND bHomeDone ,
									PT:=tPositionCfmDelayOnTime , Q=> , ET=> );

									IF ARtDelayTimer[iSignalFL1,iSignalFL2,iSignalFL3].Q THEN
									DSArmPosition.AR3sbPositionCfm[iSignalFL1,iSignalFL2,iSignalFL3] := TRUE;
									ELSE
									DSArmPosition.AR3sbPositionCfm[iSignalFL1,iSignalFL2,iSignalFL3] := FALSE;
									END_IF
								ELSE
								DSArmPosition.AR3sbPositionCfm[iSignalFL1,iSignalFL2,iSignalFL3] := FALSE;
								END_IF
							END_IF




						ELSE
							DSArmPosition.AR3sbPositionCfm[iSignalFL1,iSignalFL2,iSignalFL3] := FALSE;
							DSArmPosition.AR3sb2ndSpdEn[iSignalFL1,iSignalFL2,iSignalFL3] := FALSE;
						END_IF

					END_IF
				END_FOR
			END_IF
		END_FOR
	END_IF
END_FOR

END_FUNCTION_BLOCK

// ---- FBs/B_JKS_NewFB_V2/FBP-ArmRelated/NIUfbV2_FBPVertArmPosConfirm.TcPOU
FUNCTION_BLOCK NIUfbV2_FBPVertArmPosConfirm
VAR_INPUT
	bEnable 						: BOOL;
(*	ARiLdStnID						: INT;
	ARiUldStnID						: INT;
*)	lrCurrentVertActualPos 		: LREAL; (*From Encoder Reading*)
	iCurrentHorzZoneNo 			: INT; (*From fbFBPArmZoneConfirm Output*)
	ARDSLdZonePosOut 			: ARRAY [0..iLdStnQty] OF DSA32_StationZonePosOut; (*From fbGnrProductRecipeMemory Output*)
	ARDSStationZonePosOut 		: ARRAY [0..iStnQty] OF DSA32_StationZonePosOut; (*From fbGnrProductRecipeMemory Output*)
	ARDSUldZonePosOut 			: ARRAY [0..iUldStnQty] OF DSA32_StationZonePosOut; (*From fbGnrProductRecipeMemory Output*)



END_VAR
VAR_OUTPUT
	bVertTopTravelPosConfirm 	: BOOL;
	bVertMidTravelPosConfirm 	: BOOL;
	bVertDownPosConfirm 		: BOOL;


END_VAR
VAR
	DSBufferZonePosOut : DSA32_StationZonePosOut;
	DSEmptyZonePosOut : DSA32_StationZonePosOut;
	iBufferFL: INT;
	bHorzZoneNoFound: BOOL;
END_VAR

(*Pos Confirm Checking Start*)
IF bEnable THEN
bHorzZoneNoFound := FALSE;

	IF NOT bHorzZoneNoFound THEN
		iBufferFL := 1;
			FOR iBufferFL := 1 TO iLdStnQty DO
				IF iBufferFL >= 1 AND iBufferFL <= iLdStnQty THEN
					IF iCurrentHorzZoneNo = ARiLdStnID[iBufferFL] THEN
					DSBufferZonePosOut := ARDSLdZonePosOut[iBufferFL];
					bHorzZoneNoFound := TRUE;
					END_IF
				END_IF
			END_FOR
	END_IF

	IF NOT bHorzZoneNoFound THEN
		iBufferFL := 1;
			FOR iBufferFL := 1 TO iUldStnQty DO
				IF iBufferFL >= 1 AND iBufferFL <= iUldStnQty THEN
					IF iCurrentHorzZoneNo = ARiUldStnID[iBufferFL] THEN
					DSBufferZonePosOut := ARDSUldZonePosOut[iBufferFL];
					bHorzZoneNoFound := TRUE;
					END_IF
				END_IF
			END_FOR
	END_IF

	IF NOT bHorzZoneNoFound THEN
		iBufferFL := 1;
		iBufferFL := 1;
			FOR iBufferFL := 1 TO iStnQty DO
				IF iBufferFL >= 1 AND iBufferFL <= iStnQty THEN
					IF iCurrentHorzZoneNo = iBufferFL THEN
					DSBufferZonePosOut := ARDSStationZonePosOut[iBufferFL];
					bHorzZoneNoFound := TRUE;
					END_IF
				END_IF
			END_FOR
	END_IF


(*Generate Bit*)

	IF DSBufferZonePosOut.lrZone1StartPos > 1 AND DSBufferZonePosOut.lrZone1StartPos = lrCurrentVertActualPos THEN
	bVertTopTravelPosConfirm := TRUE;
	ELSE
	bVertTopTravelPosConfirm := FALSE;
	END_IF

	IF DSBufferZonePosOut.lrMidPos > 1 AND DSBufferZonePosOut.lrMidPos = lrCurrentVertActualPos THEN
	bVertMidTravelPosConfirm := TRUE;
	ELSE
	bVertMidTravelPosConfirm := FALSE;
	END_IF

	IF DSBufferZonePosOut.lrZone4EndPos > 1 AND DSBufferZonePosOut.lrZone4EndPos = lrCurrentVertActualPos THEN
	bVertDownPosConfirm := TRUE;
	ELSE
	bVertDownPosConfirm := FALSE;
	END_IF




END_IF






(*Reset*)
IF NOT bHorzZoneNoFound THEN
	DSBufferZonePosOut := DSEmptyZonePosOut;
END_IF

IF NOT bEnable OR iCurrentHorzZoneNo <= 0 THEN
	bVertTopTravelPosConfirm 	:= FALSE;
	bVertMidTravelPosConfirm 	:= FALSE;
	bVertDownPosConfirm 		:= FALSE;
	DSBufferZonePosOut := DSEmptyZonePosOut;

END_IF

END_FUNCTION_BLOCK

// ---- FBs/B_JKS_NewFB_V2/FBP-Function_Sub/fbAgitationCtrl.TcPOU
FUNCTION_BLOCK fbAgitationCtrl
VAR_INPUT
	bAgitationEn								: BOOL;
	lrCurrentPos								: LREAL;

END_VAR
VAR_OUTPUT
	bAgitation_in_Progress						: BOOL;
	bAgitation_Completed						: BOOL;

	bOut_InvMoveFwd							 : BOOL;
	bOut_InvMoveRwd						 : BOOL;

	bOut_InvMove2ndSpd						 : BOOL;
	rPosTargetSpdHz							 : REAL;
	lrTargetPos								: LREAL;

END_VAR
VAR_IN_OUT

	DSAgitationParameterIn		: DSPnpAgitationParameter;

END_VAR
VAR
	bPosStRE: R_TRIG;
	iStep: INT;
	iCount	: INT;
	bBtmLowRange: BOOL;
	bBtmHighRange: BOOL;
	bTopLowRange: BOOL;
	bTopHighRange: BOOL;
END_VAR

bPosStRE(CLK:= bAgitationEn , Q=> );

IF bPosStRE.Q THEN

iStep := 1;
END_IF

IF  NOT bAgitationEn  THEN
iStep := 0;
END_IF

CASE iStep OF

0:

	bAgitation_Completed := FALSE;
	bAgitation_in_Progress := FALSE;

	bOut_InvMoveFwd := FALSE;
	bOut_InvMoveRwd := FALSE;

	rPosTargetSpdHz := 0;
	lrTargetPos := 0;
	iCount := 0;

1:
	iCount := iCount + 1;

	IF iCount > DSAgitationParameterIn.iRepeatUpDownCycle THEN
		iStep := 4;
	ELSE
		iStep := 2;
	END_IF

2:
	rPosTargetSpdHz := DSAgitationParameterIn.lrAgitationSpeed;
	lrTargetPos		:= DSAgitationParameterIn.lrAgitationBtmPosition;

	IF lrCurrentPos > (DSAgitationParameterIn.lrAgitationBtmPosition-4) THEN
		bBtmLowRange := TRUE;
	ELSE
		bBtmLowRange := FALSE;
	END_IF

	IF lrCurrentPos < (DSAgitationParameterIn.lrAgitationBtmPosition+4) THEN
		bBtmHighRange	:= TRUE;
	ELSE
		bBtmHighRange	:= FALSE;
	END_IF

	IF NOT bBtmLowRange  THEN
		bOut_InvMoveFwd := TRUE;
		bOut_InvMoveRwd := FALSE;
	ELSIF NOT bBtmHighRange THEN
		bOut_InvMoveFwd := FALSE;
		bOut_InvMoveRwd := TRUE;
	ELSE
		bOut_InvMoveFwd := FALSE;
		bOut_InvMoveRwd := FALSE;
	END_IF

	IF (bBtmLowRange AND bBtmHighRange ) AND NOT bOut_InvMoveFwd AND NOT bOut_InvMoveRwd AND NOT DSAgitationParameterIn.bAgitationComplete THEN
		iStep := 3;
	END_IF

3:

	DSAgitationParameterIn.bAgitationInProgress := TRUE;

	rPosTargetSpdHz := DSAgitationParameterIn.lrAgitationSpeed;
	lrTargetPos		:= DSAgitationParameterIn.lrAgitationTopPosition;

	IF lrCurrentPos > (DSAgitationParameterIn.lrAgitationTopPosition-4) THEN
		bTopLowRange := TRUE;
	ELSE
		bTopLowRange := FALSE;
	END_IF

	IF lrCurrentPos < (DSAgitationParameterIn.lrAgitationTopPosition+4) THEN
		bTopHighRange	:= TRUE;
	ELSE
		bTopHighRange	:= FALSE;
	END_IF

	IF NOT bTopLowRange  THEN
		bOut_InvMoveFwd := TRUE;
		bOut_InvMoveRwd := FALSE;
	ELSIF NOT bTopHighRange THEN
		bOut_InvMoveFwd := FALSE;
		bOut_InvMoveRwd := TRUE;
	ELSE
		bOut_InvMoveFwd := FALSE;
		bOut_InvMoveRwd := FALSE;
	END_IF

	IF (bTopLowRange AND bTopHighRange)AND NOT bOut_InvMoveFwd AND NOT bOut_InvMoveRwd AND NOT DSAgitationParameterIn.bAgitationComplete THEN
		iStep := 1;
	END_IF

4:

		DSAgitationParameterIn.bAgitationComplete 	:= TRUE;
		bAgitation_Completed						:= TRUE;
		bAgitation_in_Progress := FALSE;

END_CASE

END_FUNCTION_BLOCK

// ---- FBs/B_JKS_NewFB_V2/FBP-Function_Sub/fbV2_DSMovementHandler.TcPOU
FUNCTION_BLOCK fbV2_DSMovementHandler
VAR_INPUT
	bCondition1 : BOOL;
	bCondition2 : BOOL;
	bCondition3 : BOOL;
	bCondition4 : BOOL;
	bCondition5 : BOOL;
	bCondition6 : BOOL;
	bCondition7 : BOOL;
	bCondition8 : BOOL;
	bCondition9 : BOOL;
	bCondition10 : BOOL;

	DSMovement1 : DS_SA_Movement;
	DSMovement2 : DS_SA_Movement;
	DSMovement3 : DS_SA_Movement;
	DSMovement4 : DS_SA_Movement;
	DSMovement5 : DS_SA_Movement;
	DSMovement6 : DS_SA_Movement;
	DSMovement7 : DS_SA_Movement;
	DSMovement8 : DS_SA_Movement;
	DSMovement9 : DS_SA_Movement;
	DSMovement10 : DS_SA_Movement;
	DSMovementDefault : DS_SA_Movement;
END_VAR
VAR_OUTPUT
	iCurrentConditionNo : INT;
	DS_Movement_Result : DS_SA_Movement;

END_VAR
VAR
END_VAR

IF bCondition1 THEN
DS_Movement_Result := DSMovement1;
iCurrentConditionNo := 1;

ELSIF bCondition2 THEN
DS_Movement_Result := DSMovement2;
iCurrentConditionNo := 2;

ELSIF bCondition3 THEN
DS_Movement_Result := DSMovement3;
iCurrentConditionNo := 3;

ELSIF bCondition4 THEN
DS_Movement_Result := DSMovement4;
iCurrentConditionNo := 4;

ELSIF bCondition5 THEN
DS_Movement_Result := DSMovement5;
iCurrentConditionNo := 5;

ELSIF bCondition6 THEN
DS_Movement_Result := DSMovement6;
iCurrentConditionNo := 6;

ELSIF bCondition7 THEN
DS_Movement_Result := DSMovement7;
iCurrentConditionNo := 7;

ELSIF bCondition8 THEN
DS_Movement_Result := DSMovement8;
iCurrentConditionNo := 8;

ELSIF bCondition9 THEN
DS_Movement_Result := DSMovement9;
iCurrentConditionNo := 9;

ELSIF bCondition10 THEN
DS_Movement_Result := DSMovement10;
iCurrentConditionNo := 10;

ELSE
DS_Movement_Result := DSMovementDefault;
iCurrentConditionNo := 0;

END_IF
;

END_FUNCTION_BLOCK

// ---- FBs/B_JKS_NewFB_V2/FBP-Function_Sub/fbV2_InvAnalogSpdCtrl.TcPOU
FUNCTION_BLOCK fbV2_InvAnalogSpdCtrl
VAR_INPUT
	bJogEn : BOOL;
	bHomeEn : BOOL;
	bPosEn : BOOL;

	rJogTargetSpdHz : REAL;
	rHomeTargetSpdHz : REAL;
	rPosTargetSpdHz : REAL;

	bEstop : BOOL;

END_VAR
VAR_IN_OUT PERSISTENT
	rHzToRawRatio : REAL;
END_VAR

VAR_OUTPUT
	bJogInProgress : BOOL;
	bHomeInProgress : BOOL;
	bPosInProgress : BOOL;

	iAnalogOutput : INT;
	rTargetHzDisplay : REAL;

END_VAR
VAR
	iStep: INT;

END_VAR

(*Lower / Higher Limit*)
IF rHzToRawRatio < 1 THEN
rHzToRawRatio := 1;
END_IF


(*Triggering*)
IF bJogEn AND NOT bEstop THEN
iStep := 1;
ELSIF bHomeEn AND NOT bEstop THEN
iStep := 2;
ELSIF bPosEn AND NOT bEstop THEN
iStep := 3;
ELSE
iStep := 0;
END_IF


(*************Process start******************)
CASE iStep OF

(*No Operation*)
0:
bJogInProgress := FALSE;
bHomeInProgress := FALSE;
bPosInProgress := FALSE;

iAnalogOutput := 0;
rTargetHzDisplay := 0;


(*Jog Operation*)
1:
bJogInProgress := TRUE;
bHomeInProgress := FALSE;
bPosInProgress := FALSE;

iAnalogOutput := REAL_TO_INT(rJogTargetSpdHz * rHzToRawRatio);
rTargetHzDisplay := rJogTargetSpdHz;




(*Home Operation*)
2:
bJogInProgress := FALSE;
bHomeInProgress := TRUE;
bPosInProgress := FALSE;

iAnalogOutput := REAL_TO_INT(rHomeTargetSpdHz * rHzToRawRatio);
rTargetHzDisplay := rHomeTargetSpdHz;




(*Positioning Operation*)
3:
bJogInProgress := FALSE;
bHomeInProgress := FALSE;
bPosInProgress := TRUE;

iAnalogOutput := REAL_TO_INT(rPosTargetSpdHz * rHzToRawRatio);
rTargetHzDisplay := rPosTargetSpdHz;


END_CASE

END_FUNCTION_BLOCK

// ---- FBs/B_JKS_NewFB_V2/FBP-Function_Sub/fbV2_InvAxisHome.TcPOU
FUNCTION_BLOCK fbV2_InvAxisHome
VAR_INPUT
	bHomeSt : BOOL;
	bHomeReset : BOOL;
	bEstop : BOOL;
	bNegativeHomingDirectionEn : BOOL;
	bPositiveHomingDirectionEn : BOOL;
	bHomeSensor : BOOL;
	bFwdOverTravelSensorNC : BOOL;
	bRwdOverTravelSensorNC : BOOL;

	rHomeHighSpeedHz : REAL;
	rHome2ndSpeedHz : REAL;

END_VAR

VAR_IN_OUT

	rDccDelayTimeSec : REAL;

END_VAR

VAR_OUTPUT
	bHomeDone : BOOL;
	bHomeBusy : BOOL;

	bOut_InvMoveFwd : BOOL;
	bOut_InvMoveRwd : BOOL;
	bOut_EncoderValueReset : BOOL;

	rHomeTargetSpdHz : REAL;
	iHomeStep: INT;

END_VAR
VAR
	bHomeStRE: R_TRIG;
	bInternalInvMoveFwd: BOOL;
	bInternalInvMoveRwd: BOOL;
	tStep12DT: TON;
	tStep22DT: TON;
	tStep32DT: TON;
END_VAR

(*Lower / Higher Limit*)
IF rDccDelayTimeSec < 0.1 THEN
rDccDelayTimeSec := 0.1;
END_IF
IF rDccDelayTimeSec > 5 THEN
rDccDelayTimeSec := 5;
END_IF

(*Timer*)
tStep12DT(IN:=iHomeStep=12 , PT:=REAL_TO_TIME(rDccDelayTimeSec*1000) , Q=> , ET=> );
tStep22DT(IN:=iHomeStep=22 , PT:=REAL_TO_TIME(rDccDelayTimeSec*1000) , Q=> , ET=> );
tStep32DT(IN:=iHomeStep=32 , PT:=REAL_TO_TIME(rDccDelayTimeSec*1000) , Q=> , ET=> );




(*Homing Control*)
bHomeStRE(CLK:=bHomeSt , Q=> );

IF bEstop OR bHomeReset OR NOT bFwdOverTravelSensorNC OR NOT bRwdOverTravelSensorNC THEN
iHomeStep := 0;
ELSIF bHomeStRE.Q AND NOT bHomeDone THEN
iHomeStep := 1;
ELSIF NOT bHomeSt AND NOT bHomeDone THEN
iHomeStep := 0;
END_IF



CASE iHomeStep OF

(*Reset or Estop*)
0:
	bHomeDone := FALSE;
	bHomeBusy := FALSE;

	bInternalInvMoveFwd := FALSE;
	bInternalInvMoveRwd := FALSE;
	bOut_EncoderValueReset := FALSE;

	rHomeTargetSpdHz := 0;


(* Homing Process*)
1:
bHomeBusy := TRUE;

IF bHomeSensor THEN
iHomeStep := 21;
ELSE
iHomeStep := 11;
END_IF





11: (*Home Search - 1st Step*)

bHomeBusy := TRUE;
bInternalInvMoveRwd := TRUE;
rHomeTargetSpdHz := rHomeHighSpeedHz;

IF bHomeSensor THEN
iHomeStep := 12;
END_IF






12: (*Home Search - 1st Step -> Delay for DCC*)

bInternalInvMoveRwd := FALSE;

IF tStep12DT.Q THEN
iHomeStep := 21;
END_IF






21: (*Home Search - 2nd Step*)

bHomeBusy := TRUE;
bInternalInvMoveFwd := TRUE;
rHomeTargetSpdHz := rHome2ndSpeedHz;

IF NOT bHomeSensor THEN
iHomeStep := 22;
END_IF







22: (*Home Search - 2nd Step -> Delay for DCC*)

bInternalInvMoveFwd := FALSE;

IF tStep22DT.Q THEN
iHomeStep := 31;
END_IF






31:(*Home Search - 3rd Step*)

bHomeBusy := TRUE;
bInternalInvMoveRwd := TRUE;
rHomeTargetSpdHz := rHome2ndSpeedHz;

IF bHomeSensor THEN
bOut_EncoderValueReset := TRUE;
iHomeStep := 32;
END_IF





32: (*Home Search - 3rd Step -> Delay for DCC*)

bInternalInvMoveRwd := FALSE;

IF tStep32DT.Q THEN
bOut_EncoderValueReset := FALSE;
iHomeStep := 40;
END_IF






40: (*Celebration - Home Done *)
bHomeBusy := FALSE;
bOut_EncoderValueReset := FALSE;
bHomeDone := TRUE;
rHomeTargetSpdHz := 0;



END_CASE



(*Direction Control*)
IF bNegativeHomingDirectionEn AND NOT bPositiveHomingDirectionEn THEN

	IF bInternalInvMoveFwd THEN
		bOut_InvMoveFwd := TRUE;
		bOut_InvMoveRwd := FALSE;
	ELSIF bInternalInvMoveRwd THEN
		bOut_InvMoveFwd := FALSE;
		bOut_InvMoveRwd := TRUE;
	ELSE
		bOut_InvMoveRwd := FALSE;
		bOut_InvMoveFwd := FALSE;
	END_IF

ELSIF NOT bNegativeHomingDirectionEn AND bPositiveHomingDirectionEn THEN

	IF bInternalInvMoveFwd THEN
		bOut_InvMoveRwd := TRUE;
		bOut_InvMoveFwd := FALSE;
	ELSIF bInternalInvMoveRwd THEN
		bOut_InvMoveRwd := FALSE;
		bOut_InvMoveFwd := TRUE;
	ELSE
		bOut_InvMoveRwd := FALSE;
		bOut_InvMoveFwd := FALSE;
	END_IF

ELSE
		bOut_InvMoveRwd := FALSE;
		bOut_InvMoveFwd := FALSE;
END_IF

END_FUNCTION_BLOCK

// ---- FBs/B_JKS_NewFB_V2/FBP-Function_Sub/fbV2_InvAxisJog.TcPOU
FUNCTION_BLOCK fbV2_InvAxisJog
VAR_INPUT
	bEstop : BOOL;
	bPositiveJogDirectionSt : BOOL;
	bNegativeJogDirectionSt : BOOL;
	bFwdOverTravelSensorNC : BOOL;
	bRwdOverTravelSensorNC : BOOL;

	rJogSpeedHz : REAL;

END_VAR

VAR_IN_OUT
	bJogEn : BOOL;

END_VAR

VAR_OUTPUT

	bOut_InvMoveFwd : BOOL;
	bOut_InvMoveRwd : BOOL;

	rJogTargetSpdHz : REAL;

END_VAR

VAR
	iStep: INT;
END_VAR

(*Jog Control*)

rJogTargetSpdHz := rJogSpeedHz;


IF bEstop THEN
iStep := 0;

ELSIF bJogEn THEN

	IF bPositiveJogDirectionSt AND bFwdOverTravelSensorNC AND NOT bNegativeJogDirectionSt   THEN
	iStep := 11;
	ELSIF bNegativeJogDirectionSt AND bRwdOverTravelSensorNC AND NOT bPositiveJogDirectionSt THEN
	iStep := 21;
	ELSE
	iStep := 1;
	END_IF

ELSE
iStep := 1;

END_IF


CASE iStep OF

(*Reset or Estop*)
0:
	bJogEn := FALSE;
	bOut_InvMoveFwd := FALSE;
	bOut_InvMoveRwd := FALSE;



(* Jog Process - Standby*)
1:

	bOut_InvMoveFwd := FALSE;
	bOut_InvMoveRwd := FALSE;



11: (*Jog Control - Forward*)

bOut_InvMoveFwd := TRUE;
bOut_InvMoveRwd := FALSE;


21: (*Jog Control - Reverse*)

bOut_InvMoveFwd := FALSE;
bOut_InvMoveRwd := TRUE;

END_CASE

END_FUNCTION_BLOCK

// ---- FBs/B_JKS_NewFB_V2/FBP-Function_Sub/fbV2_InvPosCtrl.TcPOU
FUNCTION_BLOCK fbV2_InvPosCtrl
VAR_INPUT
	bPositioningEn 							: BOOL;
	bVertMovementEn							: BOOL;
	bHorzMovementEn						: BOOL;
	b4StepsEn								: BOOL;
	lrCurrentPos								: LREAL;

	rTargetSpdHz							: REAL;
	r2ndSpdHz								: REAL;
	i2ndSpdDelayOffTimeSV_ms				: INT;

	lrPosToleranceP : ARRAY [0..3, 0..iStnQty, 0..12] OF LREAL;
	lrPosToleranceN : ARRAY [0..3, 0..iStnQty, 0..12] OF LREAL;

	DS4StepsMovement						: DS_SA_Movement;


	(*DS4StepsUpMovement					: DS_SA_Movement;*)

END_VAR

VAR_IN_OUT PERSISTENT

	DSArmPosition 					: DSV2_ArmPosition;

END_VAR
VAR_OUTPUT
	bPositioningDone : BOOL;
	bPositioningBusy : BOOL;

	bOut_InvMoveFwd : BOOL;
	bOut_InvMoveRwd : BOOL;

	bOut_InvMove2ndSpd : BOOL;
	rPosTargetSpdHz : REAL;
	lrTargetPos		: LREAL;

END_VAR
VAR
	iSFLQty: INT;
	iStep: INT;
	iTargetPosStFL1 : INT;
	iTargetPosStFL2 : INT;
	iTargetPosStFL3 : INT;

	lrBufferTargetPos: LREAL;
	iBufferFL1: INT;
	iBufferFL2: INT;
	iBufferFL3: INT;
	bPosStRE: R_TRIG;
	bPosStFE: F_TRIG;
	DSBuffer4StepsMovement: DS_SA_Movement;
	bOut_InvMove2ndSpdInternal : BOOL;

	b2ndSpdDelayOffTimer: TON;

END_VAR

(*2nd Speed Signal Delay Off*)

b2ndSpdDelayOffTimer(IN:= NOT bOut_InvMove2ndSpdInternal, PT:=INT_TO_TIME(i2ndSpdDelayOffTimeSV_ms) , Q=> , ET=> );

IF bOut_InvMove2ndSpdInternal THEN
bOut_InvMove2ndSpd := TRUE;
END_IF

IF b2ndSpdDelayOffTimer.Q THEN
bOut_InvMove2ndSpd := FALSE;
END_IF


(*Program*)
bPosStRE(CLK:=(bPositioningEn AND bVertMovementEn AND NOT bHorzMovementEn) OR (bPositioningEn AND NOT bVertMovementEn AND bHorzMovementEn) , Q=> );

IF bPosStRE.Q THEN
iStep := 1;
END_IF

IF NOT bPositioningEn OR (bVertMovementEn AND bHorzMovementEn) OR (NOT bVertMovementEn AND NOT bHorzMovementEn)  THEN
iStep := 0;
END_IF




CASE iStep OF

0:
	bPositioningDone := FALSE;
	bPositioningBusy := FALSE;

	bOut_InvMoveFwd := FALSE;
	bOut_InvMoveRwd := FALSE;

	bOut_InvMove2ndSpdInternal := FALSE;

	rPosTargetSpdHz := 0;
	lrTargetPos := 0;

	lrBufferTargetPos := 0;
	iBufferFL1 := 0;
	iBufferFL2 := 0;
	iBufferFL3 := 0;



1: (*Reset*)
(*[][][][][][][][][][][][][][][][][][][][][][][][][][][][][][][][][][][][][][][][][][][][][][][][][][][][][][][][][][][][][][][][][][][][][][][][][][][][][][][][][][][][][][][][][][][][][][][][][][][]*)

bPositioningDone := TRUE;
bPositioningBusy := FALSE;

bOut_InvMoveFwd := FALSE;
bOut_InvMoveRwd := FALSE;

bOut_InvMove2ndSpdInternal := FALSE;

iTargetPosStFL1 := 1;
lrBufferTargetPos := 0;
(*iBufferFL1 := 0;
iBufferFL2 := 0;
iBufferFL3 := 0;
*)
rPosTargetSpdHz := 0;
lrTargetPos := 0;

iStep := 2;

2: (*Search Target Pos St*)
(*[][][][][][][][][][][][][][][][][][][][][][][][][][][][][][][][][][][][][][][][][][][][][][][][][][][][][][][][][][][][][][][][][][][][][][][][][][][][][][][][][][][][][][][][][][][][][][][][][][][]*)

FOR iTargetPosStFL1 := 1 TO 3 DO
	IF iTargetPosStFL1 >= 1 AND iTargetPosStFL1 <= 3 THEN

		IF iTargetPosStFL1 = 1 THEN
		iSFLQty := iStnQty;
		ELSIF iTargetPosStFL1 = 2 THEN
		iSFLQty := iLdStnQty;
		ELSIF iTargetPosStFL1 = 3 THEN
		iSFLQty := iUldStnQty;
		END_IF

		iTargetPosStFL2 := 1;

		FOR iTargetPosStFL2 := 1 TO iSFLQty DO
			IF iTargetPosStFL2 >= 1 AND iTargetPosStFL2 <= iSFLQty THEN

				iTargetPosStFL3 := 1;

				FOR iTargetPosStFL3 := 1 TO 12 DO
					IF iTargetPosStFL3 >= 1 AND iTargetPosStFL3 <= 12 THEN

						IF DSArmPosition.AR3slrPosition[iTargetPosStFL1, iTargetPosStFL2, iTargetPosStFL3] <> 0 THEN

							IF (iTargetPosStFL3 >= 1 AND iTargetPosStFL3 <= 6 AND bVertMovementEn) OR
							(iTargetPosStFL3 >= 7 AND iTargetPosStFL3 <= 10 AND bHorzMovementEn) THEN

								IF DSArmPosition.AR3sbTargetPosSt[iTargetPosStFL1,iTargetPosStFL2,iTargetPosStFL3] AND NOT DSArmPosition.AR3sbPositionCfm[iTargetPosStFL1,iTargetPosStFL2,iTargetPosStFL3] THEN

									lrBufferTargetPos := DSArmPosition.AR3slrPosition[iTargetPosStFL1,iTargetPosStFL2,iTargetPosStFL3];
									lrTargetPos := DSArmPosition.AR3slrPosition[iTargetPosStFL1,iTargetPosStFL2,iTargetPosStFL3];
									iBufferFL1 := iTargetPosStFL1;
									iBufferFL2 := iTargetPosStFL2;
									iBufferFL3 := iTargetPosStFL3;
									iTargetPosStFL1 := 99;
									iTargetPosStFL2 := 99;
									iTargetPosStFL3 := 99;
									iStep := 3;
								END_IF

							END_IF

						END_IF

					END_IF
				END_FOR
			END_IF
		END_FOR
	END_IF
END_FOR

IF iTargetPosStFL1 > 3 AND iTargetPosStFL2 > iSFLQty AND iTargetPosStFL3 > 12 AND iStep = 2 THEN
iStep := 1;
END_IF

3: (*Determine Up or Down movement -> Swap Data if necessary*)
(*[][][][][][][][][][][][][][][][][][][][][][][][][][][][][][][][][][][][][][][][][][][][][][][][][][][][][][][][][][][][][][][][][][][][][][][][][][][][][][][][][][][][][][][][][][][][][][][][][][][]*)
IF lrTargetPos > lrCurrentPos THEN

DSBuffer4StepsMovement := DS4StepsMovement
;
(*DSBuffer4StepsMovement.lrZone1Speed		:=	DS4StepsMovement.lrZone4Speed;
DSBuffer4StepsMovement.lrZone2Speed		:=	DS4StepsMovement.lrZone3Speed;
DSBuffer4StepsMovement.lrZone3Speed		:=	DS4StepsMovement.lrZone2Speed;
DSBuffer4StepsMovement.lrZone4Speed		:=	DS4StepsMovement.lrZone1Speed;
DSBuffer4StepsMovement.lrZone1StartPos	:=	DS4StepsMovement.lrZone4EndPos;
DSBuffer4StepsMovement.lrZone2StartPos	:=	DS4StepsMovement.lrZone4StartPos;
DSBuffer4StepsMovement.lrZone3StartPos	:=	DS4StepsMovement.lrZone3StartPos;
DSBuffer4StepsMovement.lrZone4StartPos	:=	DS4StepsMovement.lrZone2StartPos;
DSBuffer4StepsMovement.lrZone4EndPos	:=	DS4StepsMovement.lrZone1StartPos;
*)

ELSE
DSBuffer4StepsMovement.lrZone1Speed		:=	DS4StepsMovement.lrZone4Speed;
DSBuffer4StepsMovement.lrZone2Speed		:=	DS4StepsMovement.lrZone3Speed;
DSBuffer4StepsMovement.lrZone3Speed		:=	DS4StepsMovement.lrZone2Speed;
DSBuffer4StepsMovement.lrZone4Speed		:=	DS4StepsMovement.lrZone1Speed;
DSBuffer4StepsMovement.lrZone1StartPos	:=	DS4StepsMovement.lrZone4EndPos;
DSBuffer4StepsMovement.lrZone2StartPos	:=	DS4StepsMovement.lrZone4StartPos;
DSBuffer4StepsMovement.lrZone3StartPos	:=	DS4StepsMovement.lrZone3StartPos;
DSBuffer4StepsMovement.lrZone4StartPos	:=	DS4StepsMovement.lrZone2StartPos;
DSBuffer4StepsMovement.lrZone4EndPos	:=	DS4StepsMovement.lrZone1StartPos;
END_IF
iStep := 4;







4: (*Move To Target Pos*)
(*[][][][][][][][][][][][][][][][][][][][][][][][][][][][][][][][][][][][][][][][][][][][][][][][][][][][][][][][][][][][][][][][][][][][][][][][][][][][][][][][][][][][][][][][][][][][][][][][][][][]*)

	bPositioningDone := FALSE;
	bPositioningBusy := TRUE;

(*Speed Control *)


	IF DSArmPosition.AR3sb2ndSpdEn[iBufferFL1,iBufferFL2,iBufferFL3]  AND iBufferFL1 >0 AND iBufferFL2 >0 AND iBufferFL3 >0 THEN
	rPosTargetSpdHz := r2ndSpdHz;
	bOut_InvMove2ndSpdInternal := TRUE;
	ELSIF NOT b4StepsEn THEN
	rPosTargetSpdHz := rTargetSpdHz;
	bOut_InvMove2ndSpdInternal := FALSE;
	ELSIF b4StepsEn THEN
	bOut_InvMove2ndSpdInternal := FALSE;



		IF lrCurrentPos(*5*) < lrBufferTargetPos(*5*)THEN
			IF DSBuffer4StepsMovement.lrZone2StartPos(*125*) > lrCurrentPos THEN
				rPosTargetSpdHz := DSBuffer4StepsMovement.lrZone1Speed;

			ELSIF DSBuffer4StepsMovement.lrZone2StartPos(*125*) <= lrCurrentPos AND DSBuffer4StepsMovement.lrZone3StartPos(*285*) > lrCurrentPos THEN
				rPosTargetSpdHz := DSBuffer4StepsMovement.lrZone2Speed;

			ELSIF DSBuffer4StepsMovement.lrZone3StartPos(*285*) <= lrCurrentPos AND DSBuffer4StepsMovement.lrZone4StartPos(*835*) > lrCurrentPos THEN
				rPosTargetSpdHz := DSBuffer4StepsMovement.lrZone3Speed;

			ELSIF DSBuffer4StepsMovement.lrZone4StartPos(*835*) <= lrCurrentPos THEN
				rPosTargetSpdHz := DSBuffer4StepsMovement.lrZone4Speed;

			END_IF

		END_IF


		IF lrCurrentPos(*5*) >= lrBufferTargetPos(*5*)THEN
				IF DSBuffer4StepsMovement.lrZone2StartPos(*835*) < lrCurrentPos THEN
				rPosTargetSpdHz := DSBuffer4StepsMovement.lrZone1Speed;

			ELSIF DSBuffer4StepsMovement.lrZone2StartPos(*835*) >= lrCurrentPos AND DSBuffer4StepsMovement.lrZone3StartPos(*285*) < lrCurrentPos THEN
				rPosTargetSpdHz := DSBuffer4StepsMovement.lrZone2Speed;

			ELSIF DSBuffer4StepsMovement.lrZone3StartPos(*285*) >= lrCurrentPos AND DSBuffer4StepsMovement.lrZone4StartPos(*125*) < lrCurrentPos THEN
				rPosTargetSpdHz := DSBuffer4StepsMovement.lrZone3Speed;

			ELSIF DSBuffer4StepsMovement.lrZone4StartPos(*125*) >= lrCurrentPos THEN
				rPosTargetSpdHz := DSBuffer4StepsMovement.lrZone4Speed;



(*			IF DSBuffer4StepsMovement.lrZone4StartPos(*835*) < lrCurrentPos THEN
						_				rPosTargetSpdHz := DSBuffer4StepsMovement.lrZone4Speed;__					
						___					
						_			ELSIF DSBuffer4StepsMovement.lrZone4StartPos(*835*) >= lrCurrentPos AND DSBuffer4StepsMovement.lrZone3StartPos(*285*) < lrCurrentPos THEN__					
						_				rPosTargetSpdHz := DSBuffer4StepsMovement.lrZone3Speed;__					
						___					
						_			ELSIF DSBuffer4StepsMovement.lrZone3StartPos(*285*) >= lrCurrentPos AND DSBuffer4StepsMovement.lrZone2StartPos(*125*) < lrCurrentPos THEN__					
						_				rPosTargetSpdHz := DSBuffer4StepsMovement.lrZone2Speed;__					
						___					
						_			ELSIF DSBuffer4StepsMovement.lrZone2StartPos(*125*) >= lrCurrentPos THEN__					
						_				rPosTargetSpdHz := DSBuffer4StepsMovement.lrZone1Speed;__					
						___					
)
			END_IF

		END_IF

(*
		IF DSBuffer4StepsMovement.lrZone1StartPos <= lrBufferTargetPos(*DSBuffer4StepsMovement.lrZone4EndPos*) THEN
			IF (*DSBuffer4StepsMovement.lrZone1StartPos <= lrCurrentPos AND*) DSBuffer4StepsMovement.lrZone2StartPos > lrCurrentPos THEN
				rPosTargetSpdHz := DSBuffer4StepsMovement.lrZone1Speed;

			ELSIF DSBuffer4StepsMovement.lrZone2StartPos <= lrCurrentPos AND DSBuffer4StepsMovement.lrZone3StartPos > lrCurrentPos THEN
				rPosTargetSpdHz := DSBuffer4StepsMovement.lrZone2Speed;

			ELSIF DSBuffer4StepsMovement.lrZone3StartPos <= lrCurrentPos AND DSBuffer4StepsMovement.lrZone4StartPos > lrCurrentPos THEN
				rPosTargetSpdHz := DSBuffer4StepsMovement.lrZone3Speed;

			ELSIF DSBuffer4StepsMovement.lrZone4StartPos <= lrCurrentPos (*AND (*DSBuffer4StepsMovement.lrZone4EndPos*)lrBufferTargetPos >= lrCurrentPos*) THEN
				rPosTargetSpdHz := DSBuffer4StepsMovement.lrZone4Speed;

			END_IF

		END_IF


		IF DSBuffer4StepsMovement.lrZone1StartPos >= lrBufferTargetPos(*DSBuffer4StepsMovement.lrZone4EndPos*) THEN
			IF (*DSBuffer4StepsMovement.lrZone1StartPos >= lrCurrentPos AND*) DSBuffer4StepsMovement.lrZone2StartPos < lrCurrentPos THEN  ;
				rPosTargetSpdHz := DSBuffer4StepsMovement.lrZone1Speed;

			ELSIF DSBuffer4StepsMovement.lrZone2StartPos >= lrCurrentPos AND DSBuffer4StepsMovement.lrZone3StartPos < lrCurrentPos THEN  ;
				rPosTargetSpdHz := DSBuffer4StepsMovement.lrZone2Speed;

			ELSIF DSBuffer4StepsMovement.lrZone3StartPos >= lrCurrentPos AND DSBuffer4StepsMovement.lrZone4StartPos < lrCurrentPos THEN  ;
				rPosTargetSpdHz := DSBuffer4StepsMovement.lrZone3Speed;

			ELSIF DSBuffer4StepsMovement.lrZone4StartPos >= lrCurrentPos (*AND (*DSBuffer4StepsMovement.lrZone4EndPos*)lrBufferTargetPos <= lrCurrentPos*) THEN  ;
				rPosTargetSpdHz := DSBuffer4StepsMovement.lrZone4Speed;

			END_IF

		END_IF

*)

(*Tobedelete- Create DS4StepsUpMovement for going Up Pos - by Lee*)
(*
		IF DS4StepsUpMovement.lrZone1StartPos >= lrBufferTargetPos(*DS4StepsUpMovement.lrZone4EndPos*) THEN
			IF DS4StepsUpMovement.lrZone1StartPos >= lrCurrentPos AND DS4StepsUpMovement.lrZone2StartPos < lrCurrentPos THEN  ;
				rPosTargetSpdHz := DS4StepsUpMovement.lrZone1Speed;

			ELSIF DS4StepsUpMovement.lrZone2StartPos >= lrCurrentPos AND DS4StepsUpMovement.lrZone3StartPos < lrCurrentPos THEN  ;
				rPosTargetSpdHz := DS4StepsUpMovement.lrZone2Speed;

			ELSIF DS4StepsUpMovement.lrZone3StartPos >= lrCurrentPos AND DS4StepsUpMovement.lrZone4StartPos < lrCurrentPos THEN  ;
				rPosTargetSpdHz := DS4StepsUpMovement.lrZone3Speed;

			ELSIF DS4StepsUpMovement.lrZone4StartPos >= lrCurrentPos AND (*DS4StepsUpMovement.lrZone4EndPos*)lrBufferTargetPos <= lrCurrentPos THEN  ;
				rPosTargetSpdHz := DS4StepsUpMovement.lrZone4Speed;

			END_IF

		END_IF
*)


	ELSE
	rPosTargetSpdHz := 0;
	bOut_InvMove2ndSpdInternal := FALSE;

	END_IF



	(*Movement Control*)
	IF lrCurrentPos > lrBufferTargetPos AND NOT DSArmPosition.AR3sbPositionCfm[iBufferFL1,iBufferFL2,iBufferFL3]
	AND NOT (lrCurrentPos >= lrPosToleranceN[iBufferFL1, iBufferFL2, iBufferFL3]  AND lrCurrentPos <= lrPosToleranceP[iBufferFL1, iBufferFL2, iBufferFL3]) THEN

	bOut_InvMoveFwd := FALSE;
	bOut_InvMoveRwd := TRUE;

	ELSIF lrCurrentPos < lrBufferTargetPos AND NOT DSArmPosition.AR3sbPositionCfm[iBufferFL1,iBufferFL2,iBufferFL3]
	AND NOT (lrCurrentPos >= lrPosToleranceN[iBufferFL1, iBufferFL2, iBufferFL3]  AND lrCurrentPos <= lrPosToleranceP[iBufferFL1, iBufferFL2, iBufferFL3]) THEN

	bOut_InvMoveFwd := TRUE;
	bOut_InvMoveRwd := FALSE;
	ELSE
	bOut_InvMoveFwd := FALSE;
	bOut_InvMoveRwd := FALSE;
	END_IF

	IF DSArmPosition.AR3sbPositionCfm[iBufferFL1,iBufferFL2,iBufferFL3] THEN
	iStep := 1;
	END_IF


END_CASE

END_FUNCTION_BLOCK

// ---- FBs/B_JKS_NewFB_V2/FBP-HMI/fbV2_ScrMapping.TcPOU
FUNCTION_BLOCK fbV2_ScrMapping

VAR_INPUT
	iCurrentScrNo : INT;
	bLoadInd : BOOL;
	bClear_SSER : BOOL;
	bClear_SSUR : BOOL;
	bCopy_SSER : BOOL;
	bCopy_SSUR : BOOL;
END_VAR

VAR_OUTPUT
END_VAR


VAR

	ScrMapCallSelfCheckRE : R_TRIG;
	iPreviousScrNo : INT;
	ScrMapCallSelfCheckHR : BOOL;
	bInvalidScrMapCallStationSequenceNo : BOOL;
	feScrMapbInvalidCallStationSequenceNo : F_TRIG;
	ScrMapCallStep : INT;
	bScrMapCallCompleted: BOOL;
	InternalTest: BOOL;
	iPreviousScrMapStnSeqRecipeNo: INT;
	ScrMapCallStepSUB: INT;
	iPreviousScrMapStnSubRecipeNo: INT;
	ScrMapCallSelfCheckHRSEQ: BOOL;
	ScrMapCallSelfCheckHRSUB: BOOL;
	iSSERFL: INT;
	iPreviousProcessTime: INT;
	iSakaiFL: INT;
	iSakaiCase: INT;
	
	bClear_SSER_RE : R_TRIG;
	bClear_SSUR_RE : R_TRIG;
	
	bCopy_SSER_FE : F_TRIG;
	bCopy_SSUR_FE : F_TRIG;
	
	
	DSV2_StationSequenceRecipeMemory_Empty : DSV2_StationSequenceRecipeMemory;
	DsSubRecipeMemory_Empty 			   : DS_SubRecipeMemory; 
	
END_VAR


VAR_IN_OUT PERSISTENT
	ScrMapStnSeqRecipe : DSV2_fbStationSequenceRecipeStore;
	ScrMapStnSubRecipe : DS_fbStationSubRecipeStore;
	ARStationStnSeqRecipe : ARRAY [0..iStnQty] OF DSV2_fbStationSequenceRecipeStore;
	ARStationStnSubRecipe : ARRAY [0..iStnQty] OF DS_fbStationSubRecipeStore;

END_VAR

(* Screen Mapping Program*)


ScrMapCallSelfCheckRE(CLK:=iCurrentScrNo <> iPreviousScrNo , Q=> );





IF (*ScrMapCallSelfCheckRE.Q*) iCurrentScrNo <> iPreviousScrNo AND NOT ScrMapCallSelfCheckHR  THEN
ScrMapCallSelfCheckHRSEQ := TRUE;
ScrMapCallSelfCheckHRSUB := TRUE;

END_IF

IF iCurrentScrNo <= 0 OR iCurrentScrNo > iStnQty THEN
bInvalidScrMapCallStationSequenceNo := TRUE;
ELSE
bInvalidScrMapCallStationSequenceNo := FALSE;
END_IF

feScrMapbInvalidCallStationSequenceNo(CLK:=bInvalidScrMapCallStationSequenceNo , Q=> );

(* Mapping for Station SEQUENCE Recipe *)
IF( ScrMapCallSelfCheckRE.Q AND NOT bInvalidScrMapCallStationSequenceNo) OR feScrMapbInvalidCallStationSequenceNo.Q THEN
ScrMapCallStep:= 1;
END_IF


CASE ScrMapCallStep OF

1:
ScrMapStnSeqRecipe := ARStationStnSeqRecipe[iCurrentScrNo];
IF NOT ScrMapCallSelfCheckHRSUB THEN
iPreviousScrNo := iCurrentScrNo;
END_IF
iPreviousScrMapStnSeqRecipeNo := ScrMapStnSeqRecipe.iStationSequenceRecipeNo;
ScrMapCallSelfCheckHRSEQ := FALSE;
ScrMapCallStep := 2;

2:
ARStationStnSeqRecipe[iCurrentScrNo] := ScrMapStnSeqRecipe;

IF iPreviousScrMapStnSeqRecipeNo <> ScrMapStnSeqRecipe.iStationSequenceRecipeNo THEN
ScrMapCallSelfCheckHRSEQ := TRUE;
ScrMapCallStep:= 1;
END_IF

END_CASE


(* Add Min Time Control - for Vacuum Tank*)
IF ScrMapStnSeqRecipe.DsStationSequenceRecipeMemory.iProcessMinTime > 0 AND ScrMapStnSeqRecipe.DsStationSequenceRecipeMemory.iCycleProcessTime > 0 THEN
	IF (ScrMapStnSeqRecipe.DsStationSequenceRecipeMemory.iProcessMinTime / ScrMapStnSeqRecipe.DsStationSequenceRecipeMemory.iCycleProcessTime) > 0
	AND (ScrMapStnSeqRecipe.DsStationSequenceRecipeMemory.iProcessMinTime >= ScrMapStnSeqRecipe.DsStationSequenceRecipeMemory.iCycleProcessTime) THEN
		ScrMapStnSeqRecipe.DsStationSequenceRecipeMemory.iCycleCalculated := (ScrMapStnSeqRecipe.DsStationSequenceRecipeMemory.iProcessMinTime / ScrMapStnSeqRecipe.DsStationSequenceRecipeMemory.iCycleProcessTime) ;
	ELSE
		ScrMapStnSeqRecipe.DsStationSequenceRecipeMemory.iCycleCalculated := 1 ;
	END_IF

ELSE

ScrMapStnSeqRecipe.DsStationSequenceRecipeMemory.iCycleCalculated := 1 ;

END_IF


ScrMapStnSeqRecipe.DsStationSequenceRecipeMemory.iCycleRemainingTime := ScrMapStnSeqRecipe.DsStationSequenceRecipeMemory.iProcessMinTime - (ScrMapStnSeqRecipe.DsStationSequenceRecipeMemory.iCycleProcessTime * ScrMapStnSeqRecipe.DsStationSequenceRecipeMemory.iCycleCalculated);






(*
iSSERFL := 1;
FOR iSSERFL := 1 TO iProductRecipeStepArrayQty DO
	IF iSSERFL >= 1 AND iSSERFL <= iProductRecipeStepArrayQty THEN
		ScrMapStnSeqRecipe.DsStationSequenceRecipeMemory.AR10iCycle[iSSERFL] := 1;
	END_IF
END_FOR
*)
ScrMapStnSeqRecipe.DsStationSequenceRecipeMemory.AR10iCycle[ScrMapStnSeqRecipe.DsStationSequenceRecipeMemory.iStepOverwriteCycle] := ScrMapStnSeqRecipe.DsStationSequenceRecipeMemory.iCycleCalculated;



(***** SAKAI REQUEST ST****)

IF iPreviousProcessTime <> ScrMapStnSubRecipe.DsSubRecipeMemory.iComCon5ProcessTimer THEN
iPreviousProcessTime := ScrMapStnSubRecipe.DsSubRecipeMemory.iComCon5ProcessTimer;
ARStationStnSubRecipe[iCurrentScrNo].DsSubRecipeMemory.iComCon5ProcessTimer := ScrMapStnSubRecipe.DsSubRecipeMemory.iComCon5ProcessTimer;
END_IF


IF iPreviousProcessTime <> ARStationStnSubRecipe[iCurrentScrNo].DsSubRecipeMemory.iComCon5ProcessTimer
AND iPreviousProcessTime = ScrMapStnSubRecipe.DsSubRecipeMemory.iComCon5ProcessTimer THEN
iSakaiCase := 1;
END_IF

CASE iSakaiCase OF
0:;

1:

ScrMapStnSubRecipe.DsSubRecipeMemory.iComCon5ProcessTimer 	:= ARStationStnSubRecipe[iCurrentScrNo].DsSubRecipeMemory.iComCon5ProcessTimer;
iPreviousProcessTime												:= ARStationStnSubRecipe[iCurrentScrNo].DsSubRecipeMemory.iComCon5ProcessTimer;
iSakaiCase := 0;

END_CASE


(***** SAKAI REQUEST END****)


(* Mapping for Station SUB Recipe *)
IF( ScrMapCallSelfCheckRE.Q AND NOT bInvalidScrMapCallStationSequenceNo) OR feScrMapbInvalidCallStationSequenceNo.Q THEN
ScrMapCallStepSUB:= 1;
END_IF


CASE ScrMapCallStepSUB OF




3:

ScrMapStnSubRecipe.DsSubRecipeMemory.iOut19SlowPullDelayTime := ARStationStnSubRecipe[iCurrentScrNo].DsSubRecipeMemory.iOut19SlowPullDelayTime;


ARStationStnSubRecipe[iCurrentScrNo] := ScrMapStnSubRecipe;

IF iPreviousScrMapStnSubRecipeNo <> ScrMapStnSubRecipe.iSubRecipeNo THEN
ScrMapCallSelfCheckHRSUB := TRUE;
ScrMapCallStepSUB:= 1;
END_IF


2:
ARStationStnSubRecipe[iCurrentScrNo] := ScrMapStnSubRecipe;
ScrMapCallStepSUB:= 3;


1:
ScrMapStnSubRecipe := ARStationStnSubRecipe[iCurrentScrNo];

iPreviousScrNo := iCurrentScrNo;
iPreviousScrMapStnSubRecipeNo := ScrMapStnSubRecipe.iSubRecipeNo;
ScrMapCallSelfCheckHRSUB := FALSE;
ScrMapCallStepSUB := 2;


END_CASE

(*Max and Min Limit*) (*SSER*)
iSSERFL := 1;
FOR iSSERFL := 1 TO iProductRecipeStepArrayQty DO
	IF iSSERFL >= 1 AND iSSERFL <= iProductRecipeStepArrayQty THEN

		IF  ScrMapStnSeqRecipe.DsStationSequenceRecipeMemory.AR10iRepeatFromStepNo[iSSERFL] > iProductRecipeStepArrayQty
		THEN ScrMapStnSeqRecipe.DsStationSequenceRecipeMemory.AR10iRepeatFromStepNo[iSSERFL] := iProductRecipeStepArrayQty;
		ELSIF ScrMapStnSeqRecipe.DsStationSequenceRecipeMemory.AR10iRepeatFromStepNo[iSSERFL] < 1
		THEN ScrMapStnSeqRecipe.DsStationSequenceRecipeMemory.AR10iRepeatFromStepNo[iSSERFL] := 1; END_IF

		IF  ScrMapStnSeqRecipe.DsStationSequenceRecipeMemory.AR10iCycle[iSSERFL] > 99
		THEN ScrMapStnSeqRecipe.DsStationSequenceRecipeMemory.AR10iCycle[iSSERFL] := 99;
		ELSIF ScrMapStnSeqRecipe.DsStationSequenceRecipeMemory.AR10iCycle[iSSERFL] < 1
		THEN ScrMapStnSeqRecipe.DsStationSequenceRecipeMemory.AR10iCycle[iSSERFL] := 1; END_IF

		IF  ScrMapStnSeqRecipe.DsStationSequenceRecipeMemory.AR10iStationSubProNo[iSSERFL] > IStationSubRecipeArrayQty
		THEN ScrMapStnSeqRecipe.DsStationSequenceRecipeMemory.AR10iStationSubProNo[iSSERFL] := IStationSubRecipeArrayQty;
		ELSIF ScrMapStnSeqRecipe.DsStationSequenceRecipeMemory.AR10iStationSubProNo[iSSERFL] < 0
		THEN ScrMapStnSeqRecipe.DsStationSequenceRecipeMemory.AR10iStationSubProNo[iSSERFL] := 0; END_IF

	END_IF
END_FOR



(*Max and Min Limit*) (*SSUR*)
IF  ScrMapStnSubRecipe.DsSubRecipeMemory.iStCon1TargetVacuumLevel > 101 THEN ScrMapStnSubRecipe.DsSubRecipeMemory.iStCon1TargetVacuumLevel := 101; ELSIF ScrMapStnSubRecipe.DsSubRecipeMemory.iStCon1TargetVacuumLevel < -101 THEN ScrMapStnSubRecipe.DsSubRecipeMemory.iStCon1TargetVacuumLevel := -101; END_IF
IF  ScrMapStnSubRecipe.DsSubRecipeMemory.iStCon2TargetPressureLevel > 101 THEN ScrMapStnSubRecipe.DsSubRecipeMemory.iStCon2TargetPressureLevel := 101; ELSIF ScrMapStnSubRecipe.DsSubRecipeMemory.iStCon2TargetPressureLevel < -101 THEN ScrMapStnSubRecipe.DsSubRecipeMemory.iStCon2TargetPressureLevel := -101; END_IF
IF  ScrMapStnSubRecipe.DsSubRecipeMemory.iStCon3TargetProTankTempLevel > 200 THEN ScrMapStnSubRecipe.DsSubRecipeMemory.iStCon3TargetProTankTempLevel := 200; ELSIF ScrMapStnSubRecipe.DsSubRecipeMemory.iStCon3TargetProTankTempLevel < 20 THEN ScrMapStnSubRecipe.DsSubRecipeMemory.iStCon3TargetProTankTempLevel := 20; END_IF
IF  ScrMapStnSubRecipe.DsSubRecipeMemory.iStCon4TargetSubTankTempLevel > 200 THEN ScrMapStnSubRecipe.DsSubRecipeMemory.iStCon4TargetSubTankTempLevel := 200; ELSIF ScrMapStnSubRecipe.DsSubRecipeMemory.iStCon4TargetSubTankTempLevel < 20 THEN ScrMapStnSubRecipe.DsSubRecipeMemory.iStCon4TargetSubTankTempLevel := 20; END_IF

IF  ScrMapStnSubRecipe.DsSubRecipeMemory.iComCon1TargetVacuumLevel > 101 THEN ScrMapStnSubRecipe.DsSubRecipeMemory.iComCon1TargetVacuumLevel := 101; ELSIF ScrMapStnSubRecipe.DsSubRecipeMemory.iComCon1TargetVacuumLevel < -101 THEN ScrMapStnSubRecipe.DsSubRecipeMemory.iComCon1TargetVacuumLevel := -101; END_IF
IF  ScrMapStnSubRecipe.DsSubRecipeMemory.iComCon2TargetPressureLevel > 101 THEN ScrMapStnSubRecipe.DsSubRecipeMemory.iComCon2TargetPressureLevel := 101; ELSIF ScrMapStnSubRecipe.DsSubRecipeMemory.iComCon2TargetPressureLevel < -101 THEN ScrMapStnSubRecipe.DsSubRecipeMemory.iComCon2TargetPressureLevel := -101; END_IF
IF  ScrMapStnSubRecipe.DsSubRecipeMemory.iComCon3TargetProTankTempLevel > 200 THEN ScrMapStnSubRecipe.DsSubRecipeMemory.iComCon3TargetProTankTempLevel := 200; ELSIF ScrMapStnSubRecipe.DsSubRecipeMemory.iComCon3TargetProTankTempLevel < 20 THEN ScrMapStnSubRecipe.DsSubRecipeMemory.iComCon3TargetProTankTempLevel := 20; END_IF
IF  ScrMapStnSubRecipe.DsSubRecipeMemory.iComCon4TargetSubTankTempLevel > 200 THEN ScrMapStnSubRecipe.DsSubRecipeMemory.iComCon4TargetSubTankTempLevel := 200; ELSIF ScrMapStnSubRecipe.DsSubRecipeMemory.iComCon4TargetSubTankTempLevel < 20 THEN ScrMapStnSubRecipe.DsSubRecipeMemory.iComCon4TargetSubTankTempLevel := 20; END_IF

IF  ScrMapStnSubRecipe.DsSubRecipeMemory.iComCon5ProcessTimer > 9999 THEN ScrMapStnSubRecipe.DsSubRecipeMemory.iComCon5ProcessTimer := 9999; ELSIF ScrMapStnSubRecipe.DsSubRecipeMemory.iComCon5ProcessTimer < 0 THEN ScrMapStnSubRecipe.DsSubRecipeMemory.iComCon5ProcessTimer := 0; END_IF

IF  ScrMapStnSubRecipe.DsSubRecipeMemory.iOut1ProTankPumpLPM > 999 THEN ScrMapStnSubRecipe.DsSubRecipeMemory.iOut1ProTankPumpLPM := 999; ELSIF ScrMapStnSubRecipe.DsSubRecipeMemory.iOut1ProTankPumpLPM < 10 THEN ScrMapStnSubRecipe.DsSubRecipeMemory.iOut1ProTankPumpLPM := 10; END_IF

IF  ScrMapStnSubRecipe.DsSubRecipeMemory.iOut2ProTankPumpHz > 300 THEN ScrMapStnSubRecipe.DsSubRecipeMemory.iOut2ProTankPumpHz := 300; ELSIF ScrMapStnSubRecipe.DsSubRecipeMemory.iOut2ProTankPumpHz < 0 THEN ScrMapStnSubRecipe.DsSubRecipeMemory.iOut2ProTankPumpHz := 0; END_IF

IF  ScrMapStnSubRecipe.DsSubRecipeMemory.iOut3ProTankBtmUsAPwrPercent > 100 THEN ScrMapStnSubRecipe.DsSubRecipeMemory.iOut3ProTankBtmUsAPwrPercent := 100; ELSIF ScrMapStnSubRecipe.DsSubRecipeMemory.iOut3ProTankBtmUsAPwrPercent < 10 THEN ScrMapStnSubRecipe.DsSubRecipeMemory.iOut3ProTankBtmUsAPwrPercent := 10; END_IF
IF  ScrMapStnSubRecipe.DsSubRecipeMemory.iOut4ProTankBtmUsBPwrPercent > 100 THEN ScrMapStnSubRecipe.DsSubRecipeMemory.iOut4ProTankBtmUsBPwrPercent := 100; ELSIF ScrMapStnSubRecipe.DsSubRecipeMemory.iOut4ProTankBtmUsBPwrPercent < 10 THEN ScrMapStnSubRecipe.DsSubRecipeMemory.iOut4ProTankBtmUsBPwrPercent := 10; END_IF
IF  ScrMapStnSubRecipe.DsSubRecipeMemory.iOut5ProTankBtmUsCPwrPercent > 100 THEN ScrMapStnSubRecipe.DsSubRecipeMemory.iOut5ProTankBtmUsCPwrPercent := 100; ELSIF ScrMapStnSubRecipe.DsSubRecipeMemory.iOut5ProTankBtmUsCPwrPercent < 10 THEN ScrMapStnSubRecipe.DsSubRecipeMemory.iOut5ProTankBtmUsCPwrPercent := 10; END_IF
IF  ScrMapStnSubRecipe.DsSubRecipeMemory.iOut6ProTankSideUsAPwrPercent > 100 THEN ScrMapStnSubRecipe.DsSubRecipeMemory.iOut6ProTankSideUsAPwrPercent := 100; ELSIF ScrMapStnSubRecipe.DsSubRecipeMemory.iOut6ProTankSideUsAPwrPercent < 10 THEN ScrMapStnSubRecipe.DsSubRecipeMemory.iOut6ProTankSideUsAPwrPercent := 10; END_IF
IF  ScrMapStnSubRecipe.DsSubRecipeMemory.iOut7ProTankSideUsBPwrPercent > 100 THEN ScrMapStnSubRecipe.DsSubRecipeMemory.iOut7ProTankSideUsBPwrPercent := 100; ELSIF ScrMapStnSubRecipe.DsSubRecipeMemory.iOut7ProTankSideUsBPwrPercent < 10 THEN ScrMapStnSubRecipe.DsSubRecipeMemory.iOut7ProTankSideUsBPwrPercent := 10; END_IF
(*
IF  ScrMapStnSubRecipe.DsSubRecipeMemory.iOut8ProTankBtmUsAkHz > 500 THEN ScrMapStnSubRecipe.DsSubRecipeMemory.iOut8ProTankBtmUsAkHz := 500; ELSIF ScrMapStnSubRecipe.DsSubRecipeMemory.iOut8ProTankBtmUsAkHz < 25 THEN ScrMapStnSubRecipe.DsSubRecipeMemory.iOut8ProTankBtmUsAkHz := 25; END_IF
IF  ScrMapStnSubRecipe.DsSubRecipeMemory.iOut9ProTankBtmUsBkHz > 500 THEN ScrMapStnSubRecipe.DsSubRecipeMemory.iOut9ProTankBtmUsBkHz := 500; ELSIF ScrMapStnSubRecipe.DsSubRecipeMemory.iOut9ProTankBtmUsBkHz < 25 THEN ScrMapStnSubRecipe.DsSubRecipeMemory.iOut9ProTankBtmUsBkHz := 25; END_IF
IF  ScrMapStnSubRecipe.DsSubRecipeMemory.iOut10ProTankBtmUsCkHz > 500 THEN ScrMapStnSubRecipe.DsSubRecipeMemory.iOut10ProTankBtmUsCkHz := 500; ELSIF ScrMapStnSubRecipe.DsSubRecipeMemory.iOut10ProTankBtmUsCkHz < 25 THEN ScrMapStnSubRecipe.DsSubRecipeMemory.iOut10ProTankBtmUsCkHz := 25; END_IF
IF  ScrMapStnSubRecipe.DsSubRecipeMemory.iOut11ProTankSideUsAkHz > 500 THEN ScrMapStnSubRecipe.DsSubRecipeMemory.iOut11ProTankSideUsAkHz := 500; ELSIF ScrMapStnSubRecipe.DsSubRecipeMemory.iOut11ProTankSideUsAkHz < 25 THEN ScrMapStnSubRecipe.DsSubRecipeMemory.iOut11ProTankSideUsAkHz := 25; END_IF
IF  ScrMapStnSubRecipe.DsSubRecipeMemory.iOut12ProTankSideUsBkHz > 500 THEN ScrMapStnSubRecipe.DsSubRecipeMemory.iOut12ProTankSideUsBkHz := 500; ELSIF ScrMapStnSubRecipe.DsSubRecipeMemory.iOut12ProTankSideUsBkHz < 25 THEN ScrMapStnSubRecipe.DsSubRecipeMemory.iOut12ProTankSideUsBkHz := 25; END_IF
*)
IF  ScrMapStnSubRecipe.DsSubRecipeMemory.iOut13ProTankBlowerHz > 300 THEN ScrMapStnSubRecipe.DsSubRecipeMemory.iOut13ProTankBlowerHz := 300; ELSIF ScrMapStnSubRecipe.DsSubRecipeMemory.iOut13ProTankBlowerHz < 40 THEN ScrMapStnSubRecipe.DsSubRecipeMemory.iOut13ProTankBlowerHz := 40; END_IF

IF  ScrMapStnSubRecipe.DsSubRecipeMemory.rOut14ProTankChangeTemperatureDegC > 150 THEN ScrMapStnSubRecipe.DsSubRecipeMemory.rOut14ProTankChangeTemperatureDegC := 150; ELSIF ScrMapStnSubRecipe.DsSubRecipeMemory.rOut14ProTankChangeTemperatureDegC < 20 THEN ScrMapStnSubRecipe.DsSubRecipeMemory.rOut14ProTankChangeTemperatureDegC := 20; END_IF
IF  ScrMapStnSubRecipe.DsSubRecipeMemory.rOut15SubTankChangeTemperatureDegC > 150 THEN ScrMapStnSubRecipe.DsSubRecipeMemory.rOut15SubTankChangeTemperatureDegC := 150; ELSIF ScrMapStnSubRecipe.DsSubRecipeMemory.rOut15SubTankChangeTemperatureDegC < 20 THEN ScrMapStnSubRecipe.DsSubRecipeMemory.rOut15SubTankChangeTemperatureDegC := 20; END_IF


IF  ScrMapStnSubRecipe.DsSubRecipeMemory.iOut16SubTankPumpLPM > 999 THEN ScrMapStnSubRecipe.DsSubRecipeMemory.iOut16SubTankPumpLPM := 999; ELSIF ScrMapStnSubRecipe.DsSubRecipeMemory.iOut16SubTankPumpLPM < 20 THEN ScrMapStnSubRecipe.DsSubRecipeMemory.iOut16SubTankPumpLPM := 20; END_IF

IF  ScrMapStnSubRecipe.DsSubRecipeMemory.iOut17SubTankPumpHz > 300 THEN ScrMapStnSubRecipe.DsSubRecipeMemory.iOut17SubTankPumpHz := 300; ELSIF ScrMapStnSubRecipe.DsSubRecipeMemory.iOut17SubTankPumpHz < 0 THEN ScrMapStnSubRecipe.DsSubRecipeMemory.iOut17SubTankPumpHz := 0; END_IF

IF  ScrMapStnSubRecipe.DsSubRecipeMemory.iOut18SlowPullVelocity > 20(*100*) THEN ScrMapStnSubRecipe.DsSubRecipeMemory.iOut18SlowPullVelocity := 20(*100*); ELSIF ScrMapStnSubRecipe.DsSubRecipeMemory.iOut18SlowPullVelocity < 1 THEN ScrMapStnSubRecipe.DsSubRecipeMemory.iOut18SlowPullVelocity := 1; END_IF
	

bClear_SSER_RE(CLK:=bClear_SSER,Q=>);

IF bClear_SSER_RE.Q THEN
ScrMapStnSeqRecipe.iCopyToSubRecipeNo					:=0;
ScrMapStnSeqRecipe.DsStationSequenceRecipeMemory 		:=DSV2_StationSequenceRecipeMemory_Empty;
ScrMapStnSeqRecipe.sStationSequenceRecipeDescription 	:= '';

END_IF

bClear_SSUR_RE(CLK:=bClear_SSUR,Q=>);

IF bClear_SSUR_RE.Q THEN
ScrMapStnSubRecipe.iCopyToSubRecipeNo	:=0;
ScrMapStnSubRecipe.DsSubRecipeMemory 	:=DsSubRecipeMemory_Empty;
ScrMapStnSubRecipe.sSubRecipeDescription 	:= '';

END_IF

bCopy_SSER_FE(CLK:=bCopy_SSER,Q=>);

IF bCopy_SSER_FE.Q THEN
ScrMapStnSeqRecipe.iCopyToSubRecipeNo	:=0;
END_IF

bCopy_SSUR_FE(CLK:=bCopy_SSUR,Q=>);

IF bCopy_SSUR_FE.Q THEN
ScrMapStnSubRecipe.iCopyToSubRecipeNo	:=0;
END_IF

END_FUNCTION_BLOCK

// ---- FBs/B_JKS_NewFB_V2/FBP-LdUldCVRelated/fbV2_Cv2zonewith2m2sCtrl.TcPOU
FUNCTION_BLOCK fbV2_Cv2zonewith2m2sCtrl
VAR_INPUT

	bEn : BOOL;
	bResetPB : BOOL;
	rConveyorPos1DelayTime_sec : REAL;
	bCvSensor1 : BOOL;
	bCvSensor2 : BOOL;

	bCvZone1BasketConfirm : BOOL;
	bCvZone2BasketConfirm : BOOL;

	bCvZone1BasketTransfer : BOOL;
	bCvZone2BasketTransfer : BOOL;

END_VAR
VAR_OUTPUT

	bUldEndReached : BOOL;
	bCvFullSignal : BOOL;

	bCvMotor1OnOff : BOOL;
	bCvMotor2OnOff : BOOL;

	bConveyorMotorOnOffAbnormal: BOOL;
END_VAR
VAR

	bZone1Enable: BOOL;

	bCvMotor2OnOff2: BOOL;
	bCvMotor2OnOff1: BOOL;
	bCvMotor1OnOff2: BOOL;
	bCvMotor1OnOff1: BOOL;

	bTimerCountdown: BOOL;
	tCountDownDelayTimer: TON;

	bResetPBRE: R_TRIG;

	tConveyorPos1DelayTimer: TON;

END_VAR

IF bCvSensor1 AND bCvSensor2 THEN

bCvFullSignal := TRUE;
ELSE
bCvFullSignal := FALSE;
END_IF

IF bCvSensor2 THEN
bUldEndReached := TRUE;
ELSE
bUldEndReached := FALSE;
END_IF

tConveyorPos1DelayTimer(IN:=bZone1Enable AND bCvSensor2 , PT:= REAL_TO_TIME(rConveyorPos1DelayTime_sec*1000) , Q=> , ET=> );


IF bEn (*AND NOT tCountDownDelayTimer.Q*) THEN

	(* Zone1 to Zone2 *)
	IF bCvSensor1 AND NOT bCvSensor2 (*AND NOT bZone2Enable*) AND ( bCvZone1BasketConfirm OR bCvZone1BasketTransfer ) AND NOT bCvZone2BasketConfirm THEN
	bZone1Enable := TRUE;
	bCvMotor1OnOff1 := TRUE;
	bCvMotor2OnOff1 := TRUE;
	END_IF

	IF tConveyorPos1DelayTimer.Q (*bZone1Enable (*AND NOT bCvSensor1 *)AND bCvSensor2*) THEN
	bZone1Enable := FALSE;
	bCvMotor1OnOff1 := FALSE;
	bCvMotor2OnOff1 := FALSE;
	END_IF

ELSE
	bCvMotor1OnOff1 := FALSE;
	bCvMotor2OnOff1 := FALSE;

	bCvMotor1OnOff2 := FALSE;
	bCvMotor2OnOff2 := FALSE;

	bZone1Enable := FALSE;

END_IF


IF bCvMotor1OnOff1 OR bCvMotor1OnOff2 THEN
bCvMotor1OnOff := TRUE;
ELSE
bCvMotor1OnOff := FALSE;
END_IF

IF bCvMotor2OnOff1 OR bCvMotor2OnOff2 THEN
bCvMotor2OnOff := TRUE;
ELSE
bCvMotor2OnOff := FALSE;
END_IF


bResetPBRE(CLK:= bResetPB , Q=> );

IF (bZone1Enable) AND ( NOT bCvSensor1 OR NOT bCvSensor2 ) AND NOT bResetPBRE.Q THEN
bTimerCountdown := TRUE;
ELSE
bTimerCountdown := FALSE;
END_IF


tCountDownDelayTimer(IN:=bTimerCountdown , PT:=t#90s , Q=> , ET=> );

IF tCountDownDelayTimer.Q THEN
bConveyorMotorOnOffAbnormal := TRUE;
END_IF

IF bConveyorMotorOnOffAbnormal AND NOT bCvZone1BasketTransfer AND NOT bCvZone2BasketTransfer THEN
bConveyorMotorOnOffAbnormal := FALSE;
END_IF

IF bResetPBRE.Q THEN
bConveyorMotorOnOffAbnormal := FALSE;
END_IF

END_FUNCTION_BLOCK

// ---- FBs/B_JKS_NewFB_V2/FBP-MTBSubFB/fbV2_MinMaxExtShift.TcPOU
FUNCTION_BLOCK fbV2_MinMaxExtShift
VAR_INPUT
	bEN: BOOL;
	bTempPushEffTime : BOOL;
	iLdProductRecipeNo : INT;
END_VAR
VAR_OUTPUT
	DSV2LdBasketMinMaxEffTime 								: DSV2_MinMaxEffTime;
END_VAR
VAR_IN_OUT
	DSV2MTBMinMaxEffTime 								: DSV2_MinMaxEffTime;
	ARDsSSERSourceMinMaxTime_Uni						: ARRAY [1..iStnQty] OF DSV2_SSERSourceMinMaxTime;

(*	AR2SiCalledRecipeTimeBlockNoCallArmTime 			: ARRAY[1..iRecipeBlockQty, 1..9] OF INT;
	AR2SiCalledRecipeTimeBlockWithCallArmTime 			: ARRAY[1..iRecipeBlockQty, 1..9] OF INT;
*)
END_VAR
VAR
	bENRE: R_TRIG;
	iStep: INT;
	iBufferProductRecipeNo: INT;
	ARiTransferStationNoEmpty		: ARRAY [0..iProductRecipeStepArrayQty] OF INT;
	ARiStnSeqRepNoEmpty	 		: ARRAY [0..iProductRecipeStepArrayQty] OF INT;
	ARiMinTimeEmpty 				: ARRAY [0..iProductRecipeStepArrayQty] OF INT;
	ARiMaxTimeEmpty 				: ARRAY [0..iProductRecipeStepArrayQty] OF INT;
	ARiEffTimeEmpty 					: ARRAY [0..iProductRecipeStepArrayQty] OF INT;

	iScanFL: INT;
END_VAR

DSV2MTBMinMaxEffTime.iProductRecipeNo := iLdProductRecipeNo;

bENRE(CLK:=bEN AND DSV2MTBMinMaxEffTime.iProductRecipeNo <> iBufferProductRecipeNo , Q=> );
IF bENRE.Q THEN
iStep := 1;
END_IF
IF NOT bEN THEN
iStep := 0;

END_IF

CASE iStep OF

0:
	DSV2MTBMinMaxEffTime.ARiTransferStationNo	:= ARiTransferStationNoEmpty		;
	DSV2MTBMinMaxEffTime.ARiStnSeqRepNo		:= ARiStnSeqRepNoEmpty	 		;
	DSV2MTBMinMaxEffTime.ARiMinTime			:= ARiMinTimeEmpty 				;
	DSV2MTBMinMaxEffTime.ARiMaxTime			:= ARiMaxTimeEmpty 				;
	DSV2MTBMinMaxEffTime.ARiEffTime			:= ARiEffTimeEmpty 				;


1:
iScanFL := 1;
	FOR iScanFL := 1 TO iProductRecipeStepArrayQty DO
		IF iScanFL >= 1 AND iScanFL <= iProductRecipeStepArrayQty THEN
			IF (DSV2MTBMinMaxEffTime.ARiTransferStationNo[iScanFL] >= 1 AND DSV2MTBMinMaxEffTime.ARiTransferStationNo[iScanFL] <= iStnQty)
			AND (DSV2MTBMinMaxEffTime.ARiStnSeqRepNo[iScanFL] >= 1 AND DSV2MTBMinMaxEffTime.ARiStnSeqRepNo[iScanFL] <= iStationSequenceRecipeArrayQty) THEN

				DSV2MTBMinMaxEffTime.ARiMinTime[iScanFL]			:= ARDsSSERSourceMinMaxTime_Uni[DSV2MTBMinMaxEffTime.ARiTransferStationNo[iScanFL]].ARiMinTime[DSV2MTBMinMaxEffTime.ARiStnSeqRepNo[iScanFL]];
				DSV2MTBMinMaxEffTime.ARiMaxTime[iScanFL]			:= ARDsSSERSourceMinMaxTime_Uni[DSV2MTBMinMaxEffTime.ARiTransferStationNo[iScanFL]].ARiMaxTime[DSV2MTBMinMaxEffTime.ARiStnSeqRepNo[iScanFL]];

				IF bTempPushEffTime THEN
					DSV2MTBMinMaxEffTime.ARiEffTime[iScanFL]		:= ARDsSSERSourceMinMaxTime_Uni[DSV2MTBMinMaxEffTime.ARiTransferStationNo[iScanFL]].ARiMinTime[DSV2MTBMinMaxEffTime.ARiStnSeqRepNo[iScanFL]];

				END_IF


			ELSE

				DSV2MTBMinMaxEffTime.ARiMinTime[iScanFL]			:= ARiMinTimeEmpty[iScanFL] 				;
				DSV2MTBMinMaxEffTime.ARiMaxTime[iScanFL]			:= ARiMaxTimeEmpty[iScanFL] 				;
				DSV2MTBMinMaxEffTime.ARiEffTime[iScanFL]			:= ARiEffTimeEmpty[iScanFL] 				;

			END_IF
		END_IF
	END_FOR

iScanFL := 2;
iBufferProductRecipeNo := DSV2MTBMinMaxEffTime.iProductRecipeNo ;
DSV2LdBasketMinMaxEffTime := DSV2MTBMinMaxEffTime;
2:; (*Completed*)


END_CASE

END_FUNCTION_BLOCK

// ---- FBs/B_JKS_NewFB_V2/FBP-MTBSubFB/fbV2_SubAnalyzeRTBEffTime.TcPOU
FUNCTION_BLOCK fbV2_SubAnalyzeRTBEffTime
VAR_INPUT
	bReset											: BOOL;
	DSV2MTBMinMaxEffTime 							: DSV2_MinMaxEffTime;
	iRTBTotalBlockQty								: INT;
END_VAR

VAR_IN_OUT
	bEn												: BOOL;
	AR2SiRecipeTimeBlockWithCallArmTime 			: ARRAY[1..iRecipeBlockQty, 1..9] OF INT;
	DSV2BasketInfo									: DSV2_BasketInfo;
(*	ARiMinTime 										: ARRAY [0..iProductRecipeStepArrayQty] OF INT;
	ARiMaxTime 										: ARRAY [0..iProductRecipeStepArrayQty] OF INT;
	ARiEffTime 										: ARRAY [0..iProductRecipeStepArrayQty] OF INT;
*)
(* RecipeTimeBlockDetail
	1 - Start Time
	2 - End Time
	3 - Stn ID
	4 - Step No (Based on Product Recipe PnP Step No)
	5 - Busy Time <Duration> = EndTime - StartTime + 1; 
	6 - Min Time (Define by User -> Process Time Per Station)
	7 - Max Time (Define by User -> For Process Tank only)
	8 - Eff Time (Final Process Time, Used on Station Timer and Call Arm Used)
	9 - BusyLink Reference 
		0		=Non
		11-19 	= BusyLinkGroupMaster No 1
		21-29 	= BusyLinkGroupMaster No 2
		=================================
		91-99 	= BusyLinkGroupMaster No 9

		111-119 	= BusyLinkGroupMaster No 1 - 1st Stn ID
		121-129 	= BusyLinkGroupMaster No 1 - 2nd Stn ID
		131-139 	= BusyLinkGroupMaster No 1 - 3rd Stn ID

		211-219 	= BusyLinkGroupMaster No 2 - 1st Stn ID
		221-229 	= BusyLinkGroupMaster No 2 - 2nd Stn ID
		231-239 	= BusyLinkGroupMaster No 2 - 3rd Stn ID

		911-919 	= BusyLinkGroupMaster No 9 - 1st Stn ID
		921-929 	= BusyLinkGroupMaster No 9 - 2nd Stn ID
		931-939 	= BusyLinkGroupMaster No 9 - 3rd Stn ID

		

*)

END_VAR



VAR_OUTPUT
	bDone : BOOL;
	iExtTime: ARRAY[1..iRecipeBlockQty] OF INT;

END_VAR

VAR
	iExtTimeEmpty: ARRAY[1..iRecipeBlockQty] OF INT;

	bResetRE: R_TRIG;
	iStep: INT;

(*	iRtbFL: INT;*)
	iRecipeCheckFL: INT;
END_VAR

VAR_INPUT


(* RecipeTimeBlockDetail
	1 - Start Time
	2 - End Time
	3 - Stn ID
	4 - Step No (Based on Product Recipe PnP Step No)
	5 - Busy Time <Duration> = EndTime - StartTime + 1; 
	6 - Min Time (Define by User -> Process Time Per Station)
	7 - Max Time (Define by User -> For Process Tank only)
	8 - Eff Time (Final Process Time, Used on Station Timer and Call Arm Used)
	9 - BusyLink Reference ( 0=Non, 1~9=BusyLinkGroupMaster No, 11-19=Group1Slave, 21-29=Group2Slave ~ 91-99=Group9Slave)
*)

END_VAR


VAR PERSISTENT


END_VAR

bResetRE(CLK:=bReset , Q=> );

IF bResetRE.Q THEN
bDone := FALSE;
iExtTime := iExtTimeEmpty;
END_IF

(*
IF NOT bEn THEN
bDone := FALSE;
END_IF
*)


IF NOT bReset AND bEn THEN
bDone := FALSE;
iExtTime := iExtTimeEmpty;

(*
CASE iStep OF

1:
*)
	IF DSV2BasketInfo.DSV2MinMaxEffTime.iProductRecipeNo >= 1 AND DSV2BasketInfo.DSV2MinMaxEffTime.iProductRecipeNo <= iProductRecipeArrayQty THEN
		DSV2BasketInfo.DSV2MinMaxEffTime.ARiStnSeqRepNo 		:= DSV2MTBMinMaxEffTime.ARiStnSeqRepNo;
		DSV2BasketInfo.DSV2MinMaxEffTime.ARiTransferStationNo 	:= DSV2MTBMinMaxEffTime.ARiTransferStationNo;
	END_IF

	iRecipeCheckFL := 1;
	IF iRecipeCheckFL>0 AND iRecipeCheckFL <= iRTBTotalBlockQty THEN
		FOR iRecipeCheckFL := 1 TO iRTBTotalBlockQty DO
			IF AR2SiRecipeTimeBlockWithCallArmTime[iRecipeCheckFL,6] > 0 THEN

				iExtTime[iRecipeCheckFL] :=
				(AR2SiRecipeTimeBlockWithCallArmTime[iRecipeCheckFL,2] - AR2SiRecipeTimeBlockWithCallArmTime[iRecipeCheckFL,1]+1) - ( AR2SiRecipeTimeBlockWithCallArmTime[iRecipeCheckFL,5]);

				AR2SiRecipeTimeBlockWithCallArmTime[iRecipeCheckFL,8] := iExtTime[iRecipeCheckFL] + AR2SiRecipeTimeBlockWithCallArmTime[iRecipeCheckFL,6];

				IF AR2SiRecipeTimeBlockWithCallArmTime[iRecipeCheckFL,9] < 100  THEN
					DSV2BasketInfo.DSV2MinMaxEffTime.ARiMinTime[AR2SiRecipeTimeBlockWithCallArmTime[iRecipeCheckFL,4]] 	:= AR2SiRecipeTimeBlockWithCallArmTime[iRecipeCheckFL,6];
					DSV2BasketInfo.DSV2MinMaxEffTime.ARiMaxTime[AR2SiRecipeTimeBlockWithCallArmTime[iRecipeCheckFL,4]] 	:= AR2SiRecipeTimeBlockWithCallArmTime[iRecipeCheckFL,7];
					DSV2BasketInfo.DSV2MinMaxEffTime.ARiEffTime[AR2SiRecipeTimeBlockWithCallArmTime[iRecipeCheckFL,4]] 	:= AR2SiRecipeTimeBlockWithCallArmTime[iRecipeCheckFL,8];
				END_IF

			END_IF
		END_FOR
	END_IF



bDone := TRUE;
bEn := FALSE;


END_IF

END_FUNCTION_BLOCK

// ---- FBs/B_JKS_NewFB_V2/FBP-MTBSubFB/fbV2_SubBusyRTBShifting.TcPOU
FUNCTION_BLOCK fbV2_SubBusyRTBShifting
VAR_INPUT
	ARiArmID: ARRAY [1..iArmQty] OF INT;
	iRTBTotalBlockQty						: INT;

END_VAR
VAR_IN_OUT

	bEn										: BOOL;
	iShiftValue								: INT;
	iCurrentRecipeBlockNo					: INT;
	AR2SiRecipeTimeBlockWithCallArmTime 	: ARRAY[1..iRecipeBlockQty, 1..9] OF INT;
(*	iPrevious2RecipeBusyBlockStart 			: INT;	(*RD1*)		(*Array "1"*)
	iPrevious2RecipeBusyBlockEnd 			: INT;	(*RD2*)		(*Array "2"*)
	iPrevious2RecipeBusyStnID	 			: INT;	(*RD2*)		(*Array "3"*)
	iPrevious1RecipeBusyBlockStart 			: INT;	(*RD1*)		(*Array "1"*)
	iPrevious1RecipeBusyBlockEnd 			: INT;	(*RD2*)		(*Array "2"*)
	iPrevious1RecipeBusyStnID	 			: INT;	(*RD2*)		(*Array "3"*)
	iCurrentRecipeBusyBlockStart 				: INT;	(*RD1*)		(*Array "1"*)
	iCurrentRecipeBusyBlockEnd 				: INT;	(*RD2*)		(*Array "2"*)
	iCurrentRecipeBusyStnID	 				: INT;	(*RD2*)		(*Array "3"*)
*)
END_VAR

VAR_OUTPUT

	bArmIDFound							: BOOL;
	bDone								: BOOL;
	iPreviousShiftValue					: INT;


END_VAR
VAR

	bEnFE: F_TRIG;

	bResetRE: R_TRIG;
	iCheckArmIDFL: INT;
	iRTBShiftFL: INT;
END_VAR

IF NOT bEn THEN
bDone := FALSE;
END_IF



IF bEn THEN
bDone := FALSE;
bArmIDFound := FALSE;

	(*Check ArmID*)
	iCheckArmIDFL := 1;
	IF iCheckArmIDFL>0 AND iCheckArmIDFL < iArmQty+1 THEN
		FOR iCheckArmIDFL := 1 TO iArmQty DO
			IF AR2SiRecipeTimeBlockWithCallArmTime[iCurrentRecipeBlockNo,3] = ARiArmID[iCheckArmIDFL] THEN
			bArmIDFound := TRUE;
			iCheckArmIDFL := iArmQty+1;
			END_IF
		END_FOR
	END_IF

	IF iCurrentRecipeBlockNo >=3 THEN

		iRTBShiftFL := iCurrentRecipeBlockNo;

		FOR iRTBShiftFL := iCurrentRecipeBlockNo TO iRTBTotalBlockQty DO
			IF iRTBShiftFL >= iCurrentRecipeBlockNo AND iRTBShiftFL <= iRTBTotalBlockQty THEN

				IF iRTBShiftFL = iCurrentRecipeBlockNo THEN

					(*If Current is Arm, Means Previous is Station, Shifting on Arm only affect the extension of Previous Station*)
					IF bArmIDFound THEN
					AR2SiRecipeTimeBlockWithCallArmTime[iRTBShiftFL-1,1] 		:= 	AR2SiRecipeTimeBlockWithCallArmTime[iRTBShiftFL-1,1];
					AR2SiRecipeTimeBlockWithCallArmTime[iRTBShiftFL-1,2] 		:= 	AR2SiRecipeTimeBlockWithCallArmTime[iRTBShiftFL-1,2] + iShiftValue;
					AR2SiRecipeTimeBlockWithCallArmTime[iRTBShiftFL-1,3]	 	:=	AR2SiRecipeTimeBlockWithCallArmTime[iRTBShiftFL-1,3];
					AR2SiRecipeTimeBlockWithCallArmTime[iRTBShiftFL,1] 		:=	AR2SiRecipeTimeBlockWithCallArmTime[iRTBShiftFL,1] + iShiftValue;
					AR2SiRecipeTimeBlockWithCallArmTime[iRTBShiftFL,2] 		:=	AR2SiRecipeTimeBlockWithCallArmTime[iRTBShiftFL,2] + iShiftValue;
					AR2SiRecipeTimeBlockWithCallArmTime[iRTBShiftFL,3]		:=	AR2SiRecipeTimeBlockWithCallArmTime[iRTBShiftFL,3];
				
				
					(*If Current is not Arm Meant its Station. Shifting on Previous 1 = Arm (Both Start and End), Also Previous2 = PreviousStation extension*)
					ELSIF AR2SiRecipeTimeBlockWithCallArmTime[iCurrentRecipeBlockNo,3] > 0  THEN
					AR2SiRecipeTimeBlockWithCallArmTime[iRTBShiftFL-2,1] 		:=	AR2SiRecipeTimeBlockWithCallArmTime[iRTBShiftFL-2,1];
					AR2SiRecipeTimeBlockWithCallArmTime[iRTBShiftFL-2,2] 		:=	AR2SiRecipeTimeBlockWithCallArmTime[iRTBShiftFL-2,2] + iShiftValue;
					AR2SiRecipeTimeBlockWithCallArmTime[iRTBShiftFL-2,3]	 	:=	AR2SiRecipeTimeBlockWithCallArmTime[iRTBShiftFL-2,3];
					AR2SiRecipeTimeBlockWithCallArmTime[iRTBShiftFL-1,1] 		:=	AR2SiRecipeTimeBlockWithCallArmTime[iRTBShiftFL-1,1] + iShiftValue;
					AR2SiRecipeTimeBlockWithCallArmTime[iRTBShiftFL-1,2] 		:=	AR2SiRecipeTimeBlockWithCallArmTime[iRTBShiftFL-1,2] + iShiftValue;
					AR2SiRecipeTimeBlockWithCallArmTime[iRTBShiftFL-1,3]		:=	AR2SiRecipeTimeBlockWithCallArmTime[iRTBShiftFL-1,3];
					AR2SiRecipeTimeBlockWithCallArmTime[iRTBShiftFL,1] 		:=	AR2SiRecipeTimeBlockWithCallArmTime[iRTBShiftFL,1] + iShiftValue;
					AR2SiRecipeTimeBlockWithCallArmTime[iRTBShiftFL,2] 		:=	AR2SiRecipeTimeBlockWithCallArmTime[iRTBShiftFL,2] + iShiftValue;
					AR2SiRecipeTimeBlockWithCallArmTime[iRTBShiftFL,3]		:=	AR2SiRecipeTimeBlockWithCallArmTime[iRTBShiftFL,3];
					END_IF

				ELSE

					AR2SiRecipeTimeBlockWithCallArmTime[iRTBShiftFL,1] 		:=	AR2SiRecipeTimeBlockWithCallArmTime[iRTBShiftFL,1] + iShiftValue;
					AR2SiRecipeTimeBlockWithCallArmTime[iRTBShiftFL,2] 		:=	AR2SiRecipeTimeBlockWithCallArmTime[iRTBShiftFL,2] + iShiftValue;
					AR2SiRecipeTimeBlockWithCallArmTime[iRTBShiftFL,3]		:=	AR2SiRecipeTimeBlockWithCallArmTime[iRTBShiftFL,3];
				END_IF
			END_IF
		END_FOR
	END_IF

bDone := TRUE;
bEn := FALSE;
iPreviousShiftValue := iShiftValue;
iShiftValue := 0;
END_IF

END_FUNCTION_BLOCK

// ---- FBs/B_JKS_NewFB_V2/FBP-MTBSubFB/fbV2_SubFreeMTBShifting.TcPOU
FUNCTION_BLOCK fbV2_SubFreeMTBShifting
VAR_INPUT
	bReset			: BOOL;
	iShiftValue		: INT;
	AR3SiSortedMasterTimeBlockFreeArm_In					: ARRAY[1..iArmQty, 1..iMasterBlockQty, 1..3] OF INT; (* fbV2_SubMTBFreeSlotGenerator*)
	AR3SiSortedMasterTimeBlockFreeStn_In 						: ARRAY[1..iStnQty, 1..iMasterBlockQty, 1..3] OF INT; (* fbV2_SubMTBFreeSlotGenerator*)
	AR3SiSortedMasterTimeBlockFreeUld_In 					: ARRAY[1..iUldStnQty, 1..iMasterBlockQty, 1..3] OF INT; (* fbV2_SubMTBFreeSlotGenerator*)

	ARiFreeSlotDataQtyArm_in									: ARRAY[1..iArmQty] OF INT; (* fbV2_SubMTBFreeSlotGenerator*)
	ARiFreeSlotDataQtyStn_In									: ARRAY[1..iStnQty] OF INT; (* fbV2_SubMTBFreeSlotGenerator*)
	ARiFreeSlotDataQtyUld_In									: ARRAY[1..iUldStnQty] OF INT; (* fbV2_SubMTBFreeSlotGenerator*)


END_VAR

VAR_IN_OUT
	bEn				: BOOL;
	AR3SiSortedMasterTimeBlockFreeArm_Out						: ARRAY[1..iArmQty, 1..iMasterBlockQty, 1..3] OF INT; (* fbV2_SubMTBFreeSlotGenerator*)
	AR3SiSortedMasterTimeBlockFreeStn_Out 						: ARRAY[1..iStnQty, 1..iMasterBlockQty, 1..3] OF INT; (* fbV2_SubMTBFreeSlotGenerator*)
	AR3SiSortedMasterTimeBlockFreeUld_Out 						: ARRAY[1..iUldStnQty, 1..iMasterBlockQty, 1..3] OF INT; (* fbV2_SubMTBFreeSlotGenerator*)

	ARiFreeSlotDataQtyArm_Out									: ARRAY[1..iArmQty] OF INT; (* fbV2_SubMTBFreeSlotGenerator*)
	ARiFreeSlotDataQtyStn_Out									: ARRAY[1..iStnQty] OF INT; (* fbV2_SubMTBFreeSlotGenerator*)
	ARiFreeSlotDataQtyUld_Out									: ARRAY[1..iUldStnQty] OF INT; (* fbV2_SubMTBFreeSlotGenerator*)
	iStep: INT;

END_VAR



VAR_OUTPUT
	bDone					 									: BOOL;
	iPreviousShiftValue											: INT;

END_VAR
VAR
	bResetRE: R_TRIG;

	iArmFL: INT;
	iStnFL: INT;
	iUldFL: INT;
	iFreeSlotFL: INT;

	AR3SiSortedMasterTimeBlockFreeArmEmpty						: ARRAY[1..iArmQty, 1..iMasterBlockQty, 1..3] OF INT; (* fbV2_SubMTBFreeSlotGenerator*)
	AR3SiSortedMasterTimeBlockFreeStnEmpty 						: ARRAY[1..iStnQty, 1..iMasterBlockQty, 1..3] OF INT; (* fbV2_SubMTBFreeSlotGenerator*)
	AR3SiSortedMasterTimeBlockFreeUldEmpty						: ARRAY[1..iUldStnQty, 1..iMasterBlockQty, 1..3] OF INT; (* fbV2_SubMTBFreeSlotGenerator*)

	ARiFreeSlotDataQtyArmEmpty									: ARRAY[1..iArmQty] OF INT; (* fbV2_SubMTBFreeSlotGenerator*)
	ARiFreeSlotDataQtyStnEmpty									: ARRAY[1..iStnQty] OF INT; (* fbV2_SubMTBFreeSlotGenerator*)
	ARiFreeSlotDataQtyUldEmpty									: ARRAY[1..iUldStnQty] OF INT; (* fbV2_SubMTBFreeSlotGenerator*)

	AR3SiSortedMasterTimeBlockFreeArmBuffer					: ARRAY[1..iArmQty, 1..iMasterBlockQty, 1..3] OF INT; (* fbV2_SubMTBFreeSlotGenerator*)
	AR3SiSortedMasterTimeBlockFreeStnBuffer 					: ARRAY[1..iStnQty, 1..iMasterBlockQty, 1..3] OF INT; (* fbV2_SubMTBFreeSlotGenerator*)
	AR3SiSortedMasterTimeBlockFreeUldBuffer 					: ARRAY[1..iUldStnQty, 1..iMasterBlockQty, 1..3] OF INT; (* fbV2_SubMTBFreeSlotGenerator*)



	iShiftFL: INT;
	iClearZeroFL: INT;
	bEnRE: R_TRIG;
END_VAR

bResetRE(CLK:=bReset , Q=> );
bEnRE(CLK:=bEn , Q=> );

IF bResetRE.Q THEN

AR3SiSortedMasterTimeBlockFreeArm_Out 		:= AR3SiSortedMasterTimeBlockFreeArmEmpty;
AR3SiSortedMasterTimeBlockFreeStn_Out 		:= AR3SiSortedMasterTimeBlockFreeStnEmpty;
AR3SiSortedMasterTimeBlockFreeUld_Out 		:= AR3SiSortedMasterTimeBlockFreeUldEmpty;

AR3SiSortedMasterTimeBlockFreeArmBuffer 		:= AR3SiSortedMasterTimeBlockFreeArmEmpty;
AR3SiSortedMasterTimeBlockFreeStnBuffer 		:= AR3SiSortedMasterTimeBlockFreeStnEmpty;
AR3SiSortedMasterTimeBlockFreeUldBuffer 		:= AR3SiSortedMasterTimeBlockFreeUldEmpty;

ARiFreeSlotDataQtyArm_Out					:= ARiFreeSlotDataQtyArmEmpty;
ARiFreeSlotDataQtyStn_Out					:= ARiFreeSlotDataQtyStnEmpty;
ARiFreeSlotDataQtyUld_Out					:= ARiFreeSlotDataQtyUldEmpty;
bDone := FALSE;

END_IF


IF NOT bEn THEN
bDone := FALSE;
END_IF



IF NOT bReset AND bEn THEN

bDone := FALSE;

(*
CASE iStep OF

1:*)




(*Data Clear*)
AR3SiSortedMasterTimeBlockFreeArm_Out 		:= AR3SiSortedMasterTimeBlockFreeArmEmpty;
AR3SiSortedMasterTimeBlockFreeStn_Out 		:= AR3SiSortedMasterTimeBlockFreeStnEmpty;
AR3SiSortedMasterTimeBlockFreeUld_Out 		:= AR3SiSortedMasterTimeBlockFreeUldEmpty;

AR3SiSortedMasterTimeBlockFreeArmBuffer 		:= AR3SiSortedMasterTimeBlockFreeArmEmpty;
AR3SiSortedMasterTimeBlockFreeStnBuffer 		:= AR3SiSortedMasterTimeBlockFreeStnEmpty;
AR3SiSortedMasterTimeBlockFreeUldBuffer 		:= AR3SiSortedMasterTimeBlockFreeUldEmpty;

ARiFreeSlotDataQtyArm_Out					:= ARiFreeSlotDataQtyArmEmpty;
ARiFreeSlotDataQtyStn_Out					:= ARiFreeSlotDataQtyStnEmpty;
ARiFreeSlotDataQtyUld_Out					:= ARiFreeSlotDataQtyUldEmpty;



(*Minus - Shifting Value*)

	iArmFL := 1;
	FOR iArmFL := 1 TO iArmQty DO
		IF iArmFL >= 1 AND iArmFL <= iArmQty THEN
		iShiftFL := 1;
			FOR iShiftFL := 1 TO iMasterBlockQty DO
				IF iShiftFL >= 1 AND iShiftFL <= iMasterBlockQty THEN

					IF AR3SiSortedMasterTimeBlockFreeArm_In[iArmFL, iShiftFL, 2] > 0 AND iShiftFL <= ARiFreeSlotDataQtyArm_in[iArmFL] THEN
					AR3SiSortedMasterTimeBlockFreeArmBuffer[iArmFL, iShiftFL, 1] := AR3SiSortedMasterTimeBlockFreeArm_In[iArmFL, iShiftFL, 1] - iShiftValue;
					AR3SiSortedMasterTimeBlockFreeArmBuffer[iArmFL, iShiftFL, 2] := AR3SiSortedMasterTimeBlockFreeArm_In[iArmFL, iShiftFL, 2] - iShiftValue;
					AR3SiSortedMasterTimeBlockFreeArmBuffer[iArmFL, iShiftFL, 3] := AR3SiSortedMasterTimeBlockFreeArm_In[iArmFL, iShiftFL, 3];
					ELSE
					AR3SiSortedMasterTimeBlockFreeArmBuffer[iArmFL, iShiftFL, 1] := 0;
					AR3SiSortedMasterTimeBlockFreeArmBuffer[iArmFL, iShiftFL, 2] := 0;
					AR3SiSortedMasterTimeBlockFreeArmBuffer[iArmFL, iShiftFL, 3] := 0;
					END_IF
				END_IF
			END_FOR
		END_IF
	END_FOR

(*Minus - Shifting Value*)

	iStnFL := 1;
	FOR iStnFL := 1 TO iStnQty DO
		IF iStnFL >= 1 AND iStnFL <= iStnQty THEN
		iShiftFL := 1;
			FOR iShiftFL := 1 TO iMasterBlockQty DO
				IF iShiftFL >= 1 AND iShiftFL <= iMasterBlockQty THEN

					IF AR3SiSortedMasterTimeBlockFreeStn_In[iStnFL, iShiftFL, 2] > 0 AND iShiftFL <= ARiFreeSlotDataQtyStn_in[iStnFL] THEN
					AR3SiSortedMasterTimeBlockFreeStnBuffer[iStnFL, iShiftFL, 1] := AR3SiSortedMasterTimeBlockFreeStn_In[iStnFL, iShiftFL, 1] - iShiftValue;
					AR3SiSortedMasterTimeBlockFreeStnBuffer[iStnFL, iShiftFL, 2] := AR3SiSortedMasterTimeBlockFreeStn_In[iStnFL, iShiftFL, 2] - iShiftValue;
					AR3SiSortedMasterTimeBlockFreeStnBuffer[iStnFL, iShiftFL, 3] := AR3SiSortedMasterTimeBlockFreeStn_In[iStnFL, iShiftFL, 3];
					ELSE
					AR3SiSortedMasterTimeBlockFreeStnBuffer[iStnFL, iShiftFL, 1] := 0;
					AR3SiSortedMasterTimeBlockFreeStnBuffer[iStnFL, iShiftFL, 2] := 0;
					AR3SiSortedMasterTimeBlockFreeStnBuffer[iStnFL, iShiftFL, 3] := 0;
					END_IF
				END_IF
			END_FOR
		END_IF
	END_FOR


(*Minus - Shifting Value*)

	iUldFL := 1;
	FOR iUldFL := 1 TO iUldStnQty DO
		IF iUldFL >= 1 AND iUldFL <= iUldStnQty THEN
		iShiftFL := 1;
			FOR iShiftFL := 1 TO iMasterBlockQty DO
				IF iShiftFL >= 1 AND iShiftFL <= iMasterBlockQty THEN

					IF AR3SiSortedMasterTimeBlockFreeUld_In[iUldFL, iShiftFL, 2] > 0 AND iShiftFL <= ARiFreeSlotDataQtyUld_in[iUldFL] THEN
					AR3SiSortedMasterTimeBlockFreeUldBuffer[iUldFL, iShiftFL, 1] := AR3SiSortedMasterTimeBlockFreeUld_In[iUldFL, iShiftFL, 1] - iShiftValue;
					AR3SiSortedMasterTimeBlockFreeUldBuffer[iUldFL, iShiftFL, 2] := AR3SiSortedMasterTimeBlockFreeUld_In[iUldFL, iShiftFL, 2] - iShiftValue;
					AR3SiSortedMasterTimeBlockFreeUldBuffer[iUldFL, iShiftFL, 3] := AR3SiSortedMasterTimeBlockFreeUld_In[iUldFL, iShiftFL, 3];
					ELSE
					AR3SiSortedMasterTimeBlockFreeUldBuffer[iUldFL, iShiftFL, 1] := 0;
					AR3SiSortedMasterTimeBlockFreeUldBuffer[iUldFL, iShiftFL, 2] := 0;
					AR3SiSortedMasterTimeBlockFreeUldBuffer[iUldFL, iShiftFL, 3] := 0;
					END_IF
				END_IF
			END_FOR
		END_IF
	END_FOR
(*
iStep := 11;

2:
*)

(*Clear Zero*)
	iArmFL := 1;
	FOR iArmFL := 1 TO iArmQty DO
		IF iArmFL >= 1 AND iArmFL <= iArmQty THEN
		iClearZeroFL := 1;
			FOR iClearZeroFL := 1 TO ARiFreeSlotDataQtyArm_in[iArmFL] DO
				IF iClearZeroFL >= 1 AND iClearZeroFL <= ARiFreeSlotDataQtyArm_in[iArmFL] THEN

					IF AR3SiSortedMasterTimeBlockFreeArmBuffer[iArmFL, iClearZeroFL, 2] <= 0 THEN
					AR3SiSortedMasterTimeBlockFreeArmBuffer[iArmFL, iClearZeroFL, 1] := 0;
					AR3SiSortedMasterTimeBlockFreeArmBuffer[iArmFL, iClearZeroFL, 2] := 0;
					AR3SiSortedMasterTimeBlockFreeArmBuffer[iArmFL, iClearZeroFL, 3] := 0;
					ELSIF AR3SiSortedMasterTimeBlockFreeArmBuffer[iArmFL, iClearZeroFL, 1] <= 0 THEN
					AR3SiSortedMasterTimeBlockFreeArmBuffer[iArmFL, iClearZeroFL, 1] := 0;
					END_IF
				END_IF
			END_FOR
		END_IF
	END_FOR


(*Clear Zero*)
	iStnFL := 1;
	FOR iStnFL := 1 TO iStnQty DO
		IF iStnFL >= 1 AND iStnFL <= iStnQty THEN
		iClearZeroFL := 1;
			FOR iClearZeroFL := 1 TO ARiFreeSlotDataQtyStn_in[iStnFL] DO
				IF iClearZeroFL >= 1 AND iClearZeroFL <= ARiFreeSlotDataQtyStn_in[iStnFL] THEN

					IF AR3SiSortedMasterTimeBlockFreeStnBuffer[iStnFL, iClearZeroFL, 2] <= 0 THEN
					AR3SiSortedMasterTimeBlockFreeStnBuffer[iStnFL, iClearZeroFL, 1] := 0;
					AR3SiSortedMasterTimeBlockFreeStnBuffer[iStnFL, iClearZeroFL, 2] := 0;
					AR3SiSortedMasterTimeBlockFreeStnBuffer[iStnFL, iClearZeroFL, 3] := 0;
					ELSIF AR3SiSortedMasterTimeBlockFreeStnBuffer[iStnFL, iClearZeroFL, 1] <= 0 THEN
					AR3SiSortedMasterTimeBlockFreeStnBuffer[iStnFL, iClearZeroFL, 1] := 0;
					END_IF
				END_IF
			END_FOR
		END_IF
	END_FOR

(*Clear Zero*)
	iUldFL := 1;
	FOR iUldFL := 1 TO iUldStnQty DO
		IF iUldFL >= 1 AND iUldFL <= iUldStnQty THEN
		iClearZeroFL := 1;
			FOR iClearZeroFL := 1 TO ARiFreeSlotDataQtyUld_in[iUldFL] DO
				IF iClearZeroFL >= 1 AND iClearZeroFL <= ARiFreeSlotDataQtyUld_in[iUldFL] THEN

					IF AR3SiSortedMasterTimeBlockFreeUldBuffer[iUldFL, iClearZeroFL, 2] <= 0 THEN
					AR3SiSortedMasterTimeBlockFreeUldBuffer[iUldFL, iClearZeroFL, 1] := 0;
					AR3SiSortedMasterTimeBlockFreeUldBuffer[iUldFL, iClearZeroFL, 2] := 0;
					AR3SiSortedMasterTimeBlockFreeUldBuffer[iUldFL, iClearZeroFL, 3] := 0;
					ELSIF AR3SiSortedMasterTimeBlockFreeUldBuffer[iUldFL, iClearZeroFL, 1] <= 0 THEN
					AR3SiSortedMasterTimeBlockFreeUldBuffer[iUldFL, iClearZeroFL, 1] := 0;
					END_IF
				END_IF
			END_FOR
		END_IF
	END_FOR

(*
iStep := 12;

3:
*)

(*fbV2_MTBConsolidateSorted - Clear Free Slot*)

	iArmFL := 1;
	FOR iArmFL := 1 TO iArmQty DO
		IF iArmFL >= 1 AND iArmFL <= iArmQty THEN
		iFreeSlotFL := 1;
		ARiFreeSlotDataQtyArm_Out[iArmFL] := 1;
			FOR iFreeSlotFL := 1 TO ARiFreeSlotDataQtyArm_in[iArmFL] DO
				IF iFreeSlotFL >= 1 AND iFreeSlotFL <= ARiFreeSlotDataQtyArm_in[iArmFL] THEN

